CASE eMachineMode OF
	MM_Stopped:
		bAllowDoorsControl := TRUE;
		sModeMask.bRun := FALSE;
		sModeMask.bDashboard := FALSE;
		sModeMask.bManual := TRUE;
		sModeMask.bInit := bLoaderDoorsLocked AND bPearlingDoorsLocked AND NOT bInError;
		sModeMask.bStop := FALSE;
		sModeMask.bPurge := FALSE;
		sModeMask.bPause := FALSE;
		bCanChangeTool := sModeMask.bInit;
		bDoChangeTool := FALSE;
		IF sModeReq.bInit THEN
			eMachineMode := MM_Init;
		END_IF
		IF sModeReq.bManual THEN
			eMachineMode := MM_Manual;
		END_IF
		IF bChangeToolReq AND  eMachineMode = MM_Stopped AND bCanChangeTool THEN
			bDoChangeTool := TRUE;
			eMachineMode := MM_Init;
		END_IF
	MM_Init :
		bAllowDoorsControl := FALSE;
		sModeMask.bRun := FALSE;
		sModeMask.bDashboard := FALSE;
		sModeMask.bManual := FALSE;
		sModeMask.bInit := FALSE;
		sModeMask.bStop := FALSE;
		sModeMask.bPurge := FALSE;
		sModeMask.bPause := FALSE;
		IF bDoChangeTool THEN
			bCanChangeTool := bBlinking;
		ELSE
			bCanChangeTool := TRUE;
			IF bChangeToolReq THEN
				bDoChangeTool := TRUE;
			END_IF
		END_IF
		CASE eStep OF
			SP_RunStp0 : (* Init TurnOver / Pearling / Utilities*)
				eCmdTurnOver := MC_Init;
				eCmdUtilities := MC_Init;
				eCmdPearling := MC_Init;
				eStep := SP_RunStp1;
			SP_RunStp1:
				IF (sMachineData.sModTurnOver.eStatus = MS_Ready) AND (sMachineData.sModPearling.eStatus = MS_Ready) AND (sMachineData.sModUtilities.eStatus = MS_Ready) THEN
					// Init Loader / Barrel / sharpen
					eCmdLoader := MC_Init;
					eCmdBarrel := MC_Init;
					eCmdSharpen := MC_Init;
					eCmdLift1 := MC_Init;
					eCmdLift2 := MC_Init;
					eCmdReject := MC_Init;
					eStep := SP_RunStp2;
				END_IF
				IF (sMachineData.sModTurnOver.eStatus = MS_Stopped) OR  (sMachineData.sModPearling.eStatus = MS_Stopped) OR  (sMachineData.sModUtilities.eStatus = MS_Stopped) THEN
					eMachineMode := MM_ForceStop;
				END_IF
			SP_RunStp2:
				IF (sMachineData.sModLoader.eStatus = MS_Ready) AND (sMachineData.sModBarrel.eStatus = MS_Ready) AND (sMachineData.sModSharpen.eStatus = MS_Ready) THEN
					eCmdTable := MC_Init;
(*					eCmdLift1 := MC_Init;
					eCmdLift2 := MC_Init;
					eCmdReject := MC_Init;*)
					eCmdVision := MC_Init;
					eStep := SP_RunStp3;
				END_IF
				IF (sMachineData.sModLoader.eStatus = MS_Stopped) OR  (sMachineData.sModBarrel.eStatus = MS_Stopped) OR  (sMachineData.sModSharpen.eStatus = MS_Stopped) THEN
					eMachineMode := MM_ForceStop;
				END_IF
			SP_RunStp3 : (* Leave Init *)
				IF bAllModuleInReady THEN
					eMachineMode := MM_Ready;
				END_IF
				IF bOneModuleInStop THEN
					eMachineMode := MM_ForceStop;
				END_IF
		END_CASE
	MM_Ready:
		bAllowDoorsControl := TRUE;
		sModeMask.bRun := bJobInProgress AND NOT bVisionInConfig;
		sModeMask.bDashboard := TRUE;
		sModeMask.bManual := TRUE;
		sModeMask.bInit := FALSE;
		sModeMask.bStop := TRUE;
		sModeMask.bPurge := FALSE;
		sModeMask.bPause := FALSE;
		IF bDoChangeTool THEN
			bCanChangeTool := bBlinking;
		ELSE
			bCanChangeTool := TRUE;
			IF bChangeToolReq THEN
				bDoChangeTool := TRUE;
			END_IF
		END_IF
		IF sModeReq.bRun THEN eMachineMode := MM_Running; END_IF
		IF sModeReq.bDashboard THEN eMachineMode := MM_Dashboard; END_IF
		IF sModeReq.bManual THEN eMachineMode := MM_Manual; END_IF
		IF sModeReq.bStop THEN eMachineMode := MM_ForceStop; END_IF
		IF bOneModuleInStop THEN
			eMachineMode := MM_ForceStop;
		END_IF
		IF bDoChangeTool THEN
			IF eMachineMode = MM_Ready THEN
				eMachineMode := MM_Dashboard;
			ELSE
				bDoChangeTool := FALSE;
			END_IF
		END_IF
		CASE eStep OF
			SP_RunStp0:
				TReadyToStopTimer(IN:= FALSE);
			SP_RunStp1:
				TReadyToStopTimer(IN:=TRUE, PT:=t#10m);
				IF TReadyToStopTimer.Q AND eMachineMode = MM_Ready THEN
					eMachineMode := MM_ForceStop;
				END_IF
		END_CASE
	MM_Running,MM_Purging :
		bAllowDoorsControl := FALSE;
		sModeMask.bRun := FALSE;
		sModeMask.bDashboard := FALSE;
		sModeMask.bManual := FALSE;
		sModeMask.bInit := FALSE;
		sModeMask.bStop := TRUE;
		sModeMask.bPurge := (eMachineMode = MM_Running) ;
		sModeMask.bPause := TRUE;
		bCanChangeTool := FALSE;
		IF sModeReq.bPause THEN eMachineMode := MM_Pausing; END_IF
		IF sModeReq.bStop THEN eMachineMode := MM_Stopping; END_IF
		IF sModeReq.bPurge THEN
			eMachineMode := MM_Purging;
			eLastMachineMode := eMachineMode;
		END_IF
		CASE eStep OF
			SP_RunStp0:
				eCmdAll := MC_Run;
				bRunInit := TRUE;
				eStep := SP_RunStp1;
			SP_RunStp1:
				IF bRunTestMode THEN
					TManagerRunTest(
						sRunData := sRunData,
						bFirstCycle := bRunInit,
						sConfigFileData := sConfigFileData,
					);
					bRunInit := FALSE;
					sProductionCmd.TRequestSample.Activate := FALSE;
					sProductionCmd.TRequestSample.Enable := FALSE;
				ELSE
					TManagerRun(
						bSimPearling := bSimPearling,
						bPurging := (eMachineMode = MM_Purging) ,
						bFirstCycle := bRunInit,
						sRunData := sRunData,
						sConfigFileData := sConfigFileData,
						sProdLot	 := sProdLot,
						bLayeringWithTwoParts := bLayeringWithTwoParts,
						bNewJob := bNewJobForRun,
						sProductionCmd := sProductionCmd,
						bDisableCleanAfterPearling := bDisableCleanAfterPearling
					);
					bRunInit := FALSE;
					bNewJobForRun := FALSE;
					IF bOneModuleInPause OR bOneModuleInReadyOrStop THEN
						bComputeMTBF := TRUE;
					END_IF
				END_IF
				IF bOneModuleInPause THEN eMachineMode := MM_Pausing; END_IF
				IF bOneModuleInReadyOrStop THEN eMachineMode := MM_Stopping; END_IF
				IF NOT bRunTestMode AND TManagerRun.bRecipeIsFinish THEN eMachineMode := MM_Stopping; END_IF
		END_CASE
	MM_Dashboard:
		bAllowDoorsControl := TRUE;
		sModeMask.bRun := FALSE;
		sModeMask.bDashboard := FALSE;
		sModeMask.bManual := FALSE;
		sModeMask.bInit := FALSE;
		sModeMask.bStop := TRUE;
		sModeMask.bPurge := FALSE;
		sModeMask.bPause := FALSE;
		IF bDoChangeTool THEN
			bCanChangeTool := bBlinking;
		ELSE
			bCanChangeTool := TRUE;
			IF bChangeToolReq THEN
				bDoChangeTool := TRUE;
			END_IF
		END_IF
		IF sModeReq.bStop THEN eMachineMode := MM_Stopping; END_IF
		CASE eStep OF
			SP_RunStp0:
				eCmdAll := MC_Run;
				eStep := SP_RunStp1;
			SP_RunStp1:
				IF bOneModuleInPause THEN eMachineMode := MM_Pausing; END_IF
				IF bOneModuleInReadyOrStop THEN eMachineMode := MM_Stopping; END_IF
		END_CASE
		IF eMachineMode <> MM_Dashboard THEN bDoChangeTool := FALSE; END_IF
	MM_Manual :
		bAllowDoorsControl := TRUE;
		sModeMask.bRun := FALSE;
		sModeMask.bDashboard := FALSE;
		sModeMask.bManual := FALSE;
		sModeMask.bInit := bLoaderDoorsLocked AND bPearlingDoorsLocked AND NOT bInError;
		sModeMask.bStop := TRUE;
		sModeMask.bPurge := FALSE;
		sModeMask.bPause := FALSE;
		bCanChangeTool := FALSE;
		IF sModeReq.bStop THEN eMachineMode := MM_Stopping; END_IF
		IF sModeReq.bInit THEN
			eMachineMode := MM_Stopping;
			bDoInitAfterStop := TRUE;
		END_IF
		CASE eStep OF
			SP_RunStp0:
				eCmdAll := MC_Manual;
				eStep := SP_RunStp1;
			SP_RunStp1:
				eStep := SP_RunStp1;
		END_CASE;
	MM_Stopping:
		bAllowDoorsControl := FALSE;
		sModeMask.bRun := FALSE;
		sModeMask.bDashboard := FALSE;
		sModeMask.bManual := FALSE;
		sModeMask.bInit := FALSE;
		sModeMask.bStop := TRUE;
		sModeMask.bPurge := FALSE;
		sModeMask.bPause := FALSE;
		bCanChangeTool := FALSE;
		CASE eStep OF
			SP_RunStp0:
				TForceStop(IN := FALSE);
				eStep := SP_RunStp1;
			SP_RunStp1:
				TForceStop(IN := TRUE, PT := TMaxStopppingTime);
				IF bAllModuleInReady THEN
					IF TManagerRun.bRecipeIsFinish THEN
						eMachineMode := MM_Stopped;
						eCmdUtilities := MC_Stop;
					ELSE
						eMachineMode := MM_Ready;
					END_IF
					bDoInitAfterStop := FALSE;
				ELSIF bAllModuleInReadyOrStop AND bOneModuleInStop THEN
					IF bDoInitAfterStop AND bLoaderDoorsLocked AND bPearlingDoorsLocked AND NOT bInError THEN
						eMachineMode := MM_Init;
					ELSE
						eMachineMode := MM_Stopped;
					END_IF
					bDoInitAfterStop := FALSE;
				ELSIF TForceStop.Q OR sModeReq.bStop  THEN
					eMachineMode := MM_ForceStop;
				END_IF
		END_CASE;
	MM_ForceStop:
		bAllowDoorsControl := FALSE;
		sModeMask.bRun := FALSE;
		sModeMask.bDashboard := FALSE;
		sModeMask.bManual := FALSE;
		sModeMask.bInit := FALSE;
		sModeMask.bStop := FALSE;
		sModeMask.bPurge := FALSE;
		sModeMask.bPause := FALSE;
		bCanChangeTool := FALSE;
		CASE eStep OF
			SP_RunStp0:
				eCmdAll := MC_Stop;
				eStep := SP_RunStp1;
			SP_RunStp1:
				IF bAllModuleInStop THEN
					IF bDoInitAfterStop AND bLoaderDoorsLocked AND bPearlingDoorsLocked AND NOT bInError THEN
						eMachineMode := MM_Init;
					ELSE
						eMachineMode := MM_Stopped;
					END_IF
					bDoInitAfterStop := FALSE;
				END_IF
		END_CASE;
	MM_Pausing:
		bAllowDoorsControl := FALSE;
		sModeMask.bRun := FALSE;
		sModeMask.bDashboard := FALSE;
		sModeMask.bManual := FALSE;
		sModeMask.bInit := FALSE;
		sModeMask.bStop := TRUE;
		sModeMask.bPurge := FALSE;
		sModeMask.bPause := FALSE;
		bCanChangeTool := FALSE;
		CASE eStep OF
			SP_RunStp0:
				TForceStop(IN := FALSE);
				eStep := SP_RunStp1;
			SP_RunStp1:
				TForceStop(IN := TRUE, PT := TMaxPausingTime);
				IF bAllModuleInPause THEN
					eMachineMode := MM_Pause;
				ELSIF TForceStop.Q OR sModeReq.bStop OR bOneModuleInReadyOrStop  THEN
					eMachineMode := MM_Stopping;
				END_IF
		END_CASE;
	MM_Pause:
		bAllowDoorsControl := TRUE;
		sModeMask.bRun := TRUE;
		sModeMask.bDashboard := FALSE;
		sModeMask.bManual := TRUE;
		sModeMask.bInit := FALSE;
		sModeMask.bStop := TRUE;
		sModeMask.bPurge := FALSE;
		sModeMask.bPause := FALSE;
		bCanChangeTool := FALSE;
		IF sModeReq.bRun THEN eMachineMode := MM_Running; END_IF
		IF sModeReq.bManual THEN eMachineMode := MM_Manual; END_IF
		IF sModeReq.bStop THEN eMachineMode := MM_Stopping; END_IF
		IF bOneModuleInReadyOrStop THEN
			eMachineMode := MM_Stopping;
		END_IF
END_CASE;

TManagerDashboard(
	bExecute := eMachineMode = MM_Dashboard AND eLastMachineMode = eMachineMode AND eStep = SP_RunStp1,
	sRunData := sRunData,
	bDoChangeTool := bDoChangeTool,
	sConfigFileData := sConfigFileData,
	sCmd := sDashboardCmd
);

bInJobMode := ((eMachineMode = MM_Running) OR (eMachineMode = MM_Purging)) AND eLastMachineMode = eMachineMode AND eStep = SP_RunStp1 AND NOT bRunTestMode;
TJobElapsedCounter(
	bRun := bInJobMode,
	bReset := FALSE,
	bSet := FALSE
	);
TMTBFCounter(
	bStart := bInJobMode,
	bReset := FALSE
	);
IF bComputeMTBF THEN
	bComputeMTBF := FALSE;
	iMTBFCounter := iMTBFCounter + 1;
	dwMTBFTotalTime := dwMTBFTotalTime + TMTBFCounter.dwSeconds;
	TMTBFCounter(
		bReset := TRUE
		);
END_IF
IF bResetMTBF THEN
	bResetMTBF := FALSE;
	dwMTBFTotalTime := 0;
	iMTBFCounter := 0;
END_IF
IF iMTBFCounter > 0 THEN
	dwMeanMTBF := dwMTBFTotalTime / INT_TO_DWORD(iMTBFCounter);
ELSE
	dwMeanMTBF := 0;
END_IF

(* Running time counters *)
TMachineOnCounter(bStart := TRUE, bReset := bResetMachineCounters);
TInProdCounter(bStart := (eMachineMode = MM_Running) OR (eMachineMode = MM_Purging), bReset := bResetMachineCounters);

(* Clear  mode requests *)
sModeReq.bStop := FALSE;
sModeReq.bInit := FALSE;
sModeReq.bManual := FALSE;
sModeReq.bRun := FALSE;
sModeReq.bPurge := FALSE;
sModeReq.bPause := FALSE;
sModeReq.bDashboard := FALSE;


IF eCmdAll<> MC_NoCmd THEN
	eCmdLoader := eCmdAll;
	eCmdTable:= eCmdAll;
	eCmdPearling := eCmdAll;
	eCmdTurnOver := eCmdAll;
	eCmdBarrel := eCmdAll;
	eCmdSharpen := eCmdAll;
	eCmdLift1 := eCmdAll;
	eCmdLift2 := eCmdAll;
	eCmdReject := eCmdAll;
	eCmdVision := eCmdAll;
	eCmdUtilities := eCmdAll;
END_IF

TWritePersistentData(
	PORT    := 852,
	START := bSavePersistent,
	MODE    := SPDM_2PASS
);

IF bNewJob  THEN
	bJobInProgress := TRUE;
	bNewJobForRun := TRUE;
	TJobElapsedCounter(
		bRun := FALSE,
		bReset := FALSE,
		bSet := TRUE,
		tSetTime := DWORD_TO_TIME(dwStartJobElapsedTime)
	);
END_IF
IF bEndOfJob THEN
	bJobInProgress := FALSE;
	TJobElapsedCounter(
		bRun := FALSE,
		bReset := TRUE,
		bSet := FALSE
	);
END_IF
TJobElapsed := TJobElapsedCounter.TElapsed;

dwJobQty := sProdLot.dLotQty;
IF eMachineMode = MM_Purging THEN
	IF C_PROD_MODE_GOOD_PART THEN
		dwJobQty := sProdLot.dGoodQty + (sProdLot.dLoadedQty - sProdLot.dProdQty);
	ELSE
		dwJobQty := sProdLot.dLoadedQty;
	END_IF
END_IF

IF sProdLot.dEstimatedPartTime*dwJobQty > TIME_TO_DWORD(TJobElapsed) THEN
	dwProdEstimatedTimeLeft := sProdLot.dEstimatedPartTime*dwJobQty - TIME_TO_DWORD(TJobElapsed);
ELSE
	dwProdEstimatedTimeLeft := 0;
END_IF

IF NOT TWritePersistentData.BUSY AND bSavePersistent THEN
	bSavePersistent := FALSE;
END_IF

IF eMachineMode <> MM_Running AND  eMachineMode <> MM_Purging THEN
	sProductionCmd.TRequestSample.Enable := FALSE;
	sProductionCmd.TRequestSample.Activate := FALSE;
END_IF


IF eMachineMode = MM_Dashboard THEN
	eManagerRunStep := TManagerDashboard.eManagerStep;
ELSE
	IF bRunTestMode THEN
		eManagerRunStep := TManagerRunTest.eManagerStep;
	ELSE
		eManagerRunStep := TManagerRun.eManagerStep;
	END_IF
END_IF

bReadyForChangeJob := (eMachineMode = MM_Stopped);
bStopRequest := (eMachineMode = MM_Stopping);
bPauseRequest := (eMachineMode = MM_Pausing);
bPearlingHead1IsUsed := (sConfigFileData.asPearlingData[PS_SUS].THead[PH_Left].nNbOfPearls > 0) OR (sConfigFileData.asPearlingData[PS_SOUS].THead[PH_Left].nNbOfPearls > 0);
bPearlingHead2IsUsed := (sConfigFileData.asPearlingData[PS_SUS].THead[PH_Right].nNbOfPearls > 0) OR (sConfigFileData.asPearlingData[PS_SOUS].THead[PH_Right].nNbOfPearls > 0);
bLayeringWithTwoParts := ((sConfigFileData.sPartData.alrPartOffsetLayering[1].lrX <> 0) OR (sConfigFileData.sPartData.alrPartOffsetLayering[1].lrY <> 0));
bConfigError := TManagerRun.bConfigError;

(* MDE option *)
IF bFillMDE THEN
	(* Update MDE *)
	TMDEData.dwPceGood := sMachineData.sCounter.sProd.dGood;
	TMDEData.dwPceBad := sMachineData.sCounter.sProd.dTotal  - TMDEData.dwPceGood;
	
	(* MDE status *)
	IF bInError THEN
		TMDEData.iStatus := MDE_Alarm;
	ELSIF (eMachineMode = MM_Running) THEN
		TMDEData.iStatus := MDE_Production;
	ELSIF (eMachineMode = MM_Manual) THEN
		TMDEData.iStatus := MDE_Maintenance;
	ELSE
		TMDEData.iStatus := MDE_Standby;
	END_IF
	(* MDE alarm *)
	TMDEData.iPertCode := iMDEAlarm;
END_IF

END_FUNCTION_BLOCK

// ---- POUs/utils/HandleErrors.TcPOU
FUNCTION_BLOCK HandleErrors
VAR_INPUT
	bEnable					: BOOL;
(*	bUsingLeft				: BOOL;
	bUsingRight				: BOOL;*)
	abErrorsTable			: ARRAY[0..C_MAX_NB_OF_ERRORS] OF BOOL;
END_VAR
VAR_OUTPUT
	bInError					: BOOL;
	bInWarning				: BOOL;
	iMDEAlarm				: INT;
END_VAR
VAR_IN_OUT
END_VAR
VAR
END_VAR

bInError :=
	abErrorsTable[ERR_Manager]
	OR abErrorsTable[ERR_EmergencyStop]
	OR abErrorsTable[ERR_AirPressure]
	OR abErrorsTable[ERR_24VPowerSupply]
	OR abErrorsTable[ERR_48VPowerSupply]
	OR abErrorsTable[ERR_DrivesAreOFF]
	OR abErrorsTable[ERR_Aspiration]
	OR abErrorsTable[ERR_LoaderAxisX]
	OR abErrorsTable[ERR_LoaderAxisY]
	OR abErrorsTable[ERR_LoaderAxisZ1]
	OR abErrorsTable[ERR_LoaderAxisZ2]
	OR abErrorsTable[ERR_LoaderAxisTheta]
	OR abErrorsTable[ERR_LoaderHead1Vacuum]
	OR abErrorsTable[ERR_LoaderHead2Vacuum]
	OR abErrorsTable[ERR_LoaderJack]
	OR abErrorsTable[ERR_LoaderPlateVacuum]
	OR abErrorsTable[ERR_LoaderVision]
	OR abErrorsTable[ERR_LoaderNoPartTaken]
	OR abErrorsTable[ERR_Lift1Drv]
	OR abErrorsTable[ERR_Lift2Drv]
	OR abErrorsTable[ERR_BarrelAxis]
	OR abErrorsTable[ERR_BarrelJack]
	OR abErrorsTable[ERR_BarrelIndex]
	OR abErrorsTable[ERR_BarrelStickNotTaken]
	OR abErrorsTable[ERR_BarrelEmpty]
	OR abErrorsTable[ERR_PearlingAxisX]
	OR abErrorsTable[ERR_PearlingAxisY]
	OR abErrorsTable[ERR_PearlingAxisZ1]
	OR abErrorsTable[ERR_PearlingAxisZ2]
	OR abErrorsTable[ERR_PearlingSpindle1]
	OR abErrorsTable[ERR_PearlingSpindle2]
	OR abErrorsTable[ERR_PearlingGripper1]
	OR abErrorsTable[ERR_PearlingGripper2]
	OR abErrorsTable[ERR_PearlingMCR]
	OR abErrorsTable[ERR_PearlingSecurity]
	OR abErrorsTable[ERR_TableAxis]
	OR abErrorsTable[ERR_TablePearlingAspiration]
	OR abErrorsTable[ERR_TableJack]
	OR abErrorsTable[ERR_TablePos1Vacuum]
	OR abErrorsTable[ERR_TablePos2Vacuum]
	OR abErrorsTable[ERR_TablePos3Vacuum]
	OR abErrorsTable[ERR_TablePos4Vacuum]
	OR abErrorsTable[ERR_TableVacuum4Rotation]
	OR abErrorsTable[ERR_PearlingMotor1]
	OR abErrorsTable[ERR_PearlingMotor2]
	OR abErrorsTable[ERR_PearlingCurrent1]
	OR abErrorsTable[ERR_PearlingCurrent2]
	OR abErrorsTable[ERR_BrushAxis]
	OR abErrorsTable[ERR_SharpenAxis]
	OR abErrorsTable[ERR_SharpenTape]
	OR abErrorsTable[ERR_TurnOverAxis]
	OR abErrorsTable[ERR_TurnOverJack]
	OR abErrorsTable[ERR_TurnOverArmVacuum]
	OR abErrorsTable[ERR_TurnOverFixVacuum]
	OR abErrorsTable[ERR_VisionNotReady]
	OR abErrorsTable[ERR_VisionNotConnected]
	OR abErrorsTable[ERR_Vacuum]
	OR abErrorsTable[ERR_LoaderZSensorOutOfRange]
	OR abErrorsTable[ERR_RejectDrawerOpened]
	OR abErrorsTable[ERR_ConfigNotUsable]
	OR abErrorsTable[ERR_Lift1PlateLock]
	OR abErrorsTable[ERR_Lift1DrawerLock]
	OR abErrorsTable[ERR_Lift2PlateLock]
	OR abErrorsTable[ERR_Lift2DrawerLock]
	OR abErrorsTable[ERR_TableCleanBrush]
	
;

bInWarning :=
	abErrorsTable[W_LoaderDoorsNotClosed]
	OR abErrorsTable[W_PearlingDoorsNotClosed]
	OR abErrorsTable[W_NoPowerOnV1]
	OR abErrorsTable[W_DoorsNotLocked]
	OR abErrorsTable[W_LoaderSamplesReady]
	OR abErrorsTable[W_RejectChangePlate]
	OR abErrorsTable[W_Lift1NeedPlate]
	OR abErrorsTable[W_Lift2NeedPlate]
	OR abErrorsTable[W_Lift1DrawerNotInPos]
	OR abErrorsTable[W_Lift2DrawerNotInPos]
	OR abErrorsTable[W_RejectDrawerNotInPos]
	OR abErrorsTable[W_RejectPlateNotInPos]
	OR abErrorsTable[W_BarrelNeedArea1Stick]
	OR abErrorsTable[W_BarrelNeedArea2Stick]
	OR abErrorsTable[W_BarrelNeedArea3Stick]
	OR abErrorsTable[W_BarrelNeedArea4Stick]
	OR abErrorsTable[W_JobPurged]
	OR abErrorsTable[W_LoaderPartsOnPlate]
	OR abErrorsTable[W_VisionInSimulation]
	OR abErrorsTable[W_Lift1BadPlate]
	OR abErrorsTable[W_PearlingLeftStickBroken]
	OR abErrorsTable[W_PearlingRightStickBroken]
	OR abErrorsTable[W_PearlingWeight1OutOfTolerance]
	OR abErrorsTable[W_PearlingWeight2OutOfTolerance]
	OR abErrorsTable[W_PearlingLeftSpindleUsed]
	OR abErrorsTable[W_PearlingRightSpindleUsed]
	OR abErrorsTable[W_PearlingLeftMotorUsed]
	OR abErrorsTable[W_PearlingRightMotorUsed]
	OR abErrorsTable[W_PearlingLeftSpindleLimit]
	OR abErrorsTable[W_PearlingRightSpindleLimit]
	OR abErrorsTable[W_PearlingLeftSpindleHeat]
	OR abErrorsTable[W_PearlingRightSpindleHeat]
;
(* Handle TMDE error status *)
IF bInError THEN
	(* Update alarm status only if not already set *)
	IF (iMDEAlarm = 2900) OR (iMDEAlarm = 0) THEN
		(* Define code depending on alarm *)
		IF abErrorsTable[ERR_ConfigNotUsable]
				OR abErrorsTable[ERR_Aspiration]
				OR abErrorsTable[ERR_VisionNotReady]
				OR abErrorsTable[ERR_VisionNotConnected]
			THEN
			iMDEAlarm := 2010; 		(* General alarm*)
		ELSIF abErrorsTable[ERR_24VPowerSupply]
				OR abErrorsTable[ERR_48VPowerSupply]
				OR abErrorsTable[ERR_DrivesAreOFF]  THEN
			iMDEAlarm := 2020; 		(* Electrial alarm*)
		ELSIF abErrorsTable[ERR_LoaderAxisX]
				OR abErrorsTable[ERR_LoaderAxisY]
				OR abErrorsTable[ERR_LoaderAxisZ1]
				OR abErrorsTable[ERR_LoaderAxisZ2]
				OR abErrorsTable[ERR_LoaderAxisTheta]
				OR abErrorsTable[ERR_Lift1Drv]
				OR abErrorsTable[ERR_Lift2Drv]
				OR abErrorsTable[ERR_PearlingAxisX]
				OR abErrorsTable[ERR_PearlingAxisY]
				OR abErrorsTable[ERR_PearlingAxisZ1]
				OR abErrorsTable[ERR_PearlingAxisZ2]
				OR abErrorsTable[ERR_BarrelAxis]
				OR abErrorsTable[ERR_TableAxis]
				OR abErrorsTable[ERR_SharpenAxis]
				OR abErrorsTable[ERR_TurnOverAxis]
				OR abErrorsTable[ERR_BrushAxis]
				THEN
			iMDEAlarm := 2021; 		(* Motor alarm*)
		ELSIF abErrorsTable[ERR_RejectDrawerOpened]
				OR abErrorsTable[ERR_PearlingSecurity]
				OR abErrorsTable[ERR_TablePearlingAspiration]
				OR abErrorsTable[ERR_TableJack]
				OR abErrorsTable[ERR_BarrelJack]
				OR abErrorsTable[ERR_BarrelIndex]
				OR abErrorsTable[ERR_TurnOverJack]
				OR abErrorsTable[ERR_LoaderZSensorOutOfRange]
				OR abErrorsTable[ERR_LoaderJack]
				OR abErrorsTable[ERR_Lift1PlateLock]
				OR abErrorsTable[ERR_Lift1DrawerLock]
				OR abErrorsTable[ERR_Lift2PlateLock]
				OR abErrorsTable[ERR_Lift2DrawerLock]
				OR abErrorsTable[ERR_TableCleanBrush]
				THEN
			iMDEAlarm := 2040; 		(* Machine security alarm*)
		ELSIF abErrorsTable[ERR_EmergencyStop]
				THEN
			iMDEAlarm := 2050; 		(* Human security alarm*)
		ELSIF abErrorsTable[ERR_PearlingMCR]
				OR abErrorsTable[ERR_PearlingGripper1]
				OR abErrorsTable[ERR_PearlingGripper2]
				OR abErrorsTable[ERR_PearlingSpindle1]
				OR abErrorsTable[ERR_PearlingSpindle2]
				OR abErrorsTable[ERR_SharpenTape]
				THEN
			iMDEAlarm := 2060; 		(* General tool alarm*)
		ELSIF	abErrorsTable[ERR_AirPressure]
				THEN
			iMDEAlarm := 2070; 		(* Pneumatics alarm*)
		ELSIF FALSE THEN
			iMDEAlarm := 2100; 		(* Power down alarm*)
		ELSIF FALSE THEN
			iMDEAlarm := 2101; 		(* Init alarm*)
		ELSIF FALSE THEN
			iMDEAlarm := 2102; 		(* Warming alarm*)
		ELSIF FALSE THEN
			iMDEAlarm := 2103; 		(* Ready for prod alarm*)
		ELSIF abErrorsTable[ERR_BarrelEmpty] THEN
			iMDEAlarm := 2110; 		(* Material supply alarm*)
		ELSIF FALSE THEN
			iMDEAlarm := 2121; 		(* NbOfParts reached alarm*)
		ELSIF abErrorsTable[ERR_LoaderHead1Vacuum]
				OR abErrorsTable[ERR_LoaderHead2Vacuum]
				OR abErrorsTable[ERR_TablePos1Vacuum]
				OR abErrorsTable[ERR_TablePos2Vacuum]
				OR abErrorsTable[ERR_TablePos3Vacuum]
				OR abErrorsTable[ERR_TablePos4Vacuum]
				OR abErrorsTable[ERR_TurnOverArmVacuum]
				OR abErrorsTable[ERR_TurnOverFixVacuum]
				OR abErrorsTable[ERR_TableVacuum4Rotation]
				OR abErrorsTable[ERR_PearlingMotor1]
				OR abErrorsTable[ERR_PearlingMotor2]
				OR abErrorsTable[ERR_PearlingCurrent1]
				OR abErrorsTable[ERR_PearlingCurrent2]
				OR abErrorsTable[ERR_BarrelStickNotTaken]
				OR abErrorsTable[ERR_LoaderPlateVacuum]
				OR abErrorsTable[ERR_Vacuum]
				THEN
			iMDEAlarm := 2200; 		(* Process alarm*)
		ELSIF FALSE THEN
			iMDEAlarm := 2312; 		(* Tools alarm*)
		ELSE
			iMDEAlarm := 2010; 		(* By default general alarm*)
		END_IF
	END_IF
ELSIF binWarning THEN
	iMDEAlarm := 2900;
ELSE
	iMDEAlarm := 0;
END_IF

END_FUNCTION_BLOCK

// ---- POUs/utils/TBlink.TcPOU
FUNCTION_BLOCK TBlink
VAR_INPUT
	bEnable			: BOOL;
	tOnPeriod		: TIME		:= t#500ms;
	tOffPeriod		: TIME		:= t#500ms;
END_VAR
VAR_OUTPUT
	bBlink			: BOOL;
END_VAR
VAR
	TBlinker			: TON;
(*	bBlinkOn			: BOOL;*)
	CurrentPeriod		: TIME		:= t#10ms;
END_VAR

IF bEnable THEN
	TBlinker(IN := TRUE,PT := CurrentPeriod);
ELSE
	TBlinker(IN := FALSE);
END_IF

IF bBlink AND TBlinker.Q THEN
	bBlink := FALSE;
	CurrentPeriod := tOffPeriod;
	TBlinker(IN := FALSE);
ELSIF NOT bBlink AND TBlinker.Q THEN
	bBlink := TRUE;
	CurrentPeriod := tOnPeriod;
	TBlinker(IN := FALSE);
END_IF

END_FUNCTION_BLOCK

// ---- POUs/Manager/ManagerDashboard.TcPOU
FUNCTION_BLOCK ManagerDashboard
VAR_INPUT
	sConfigFileData			: TConfigFileData;
(*	bFirstCycle				: BOOL;*)
	bExecute				: BOOL;
END_VAR
VAR_OUTPUT
END_VAR
VAR_IN_OUT
	bDoChangeTool			: BOOL;
	sRunData				: TRunData;
	sCmd					: TDashboardCmd;
END_VAR
VAR
	eManagerStep			: TModuleSteps := SP_RunStp0;
	bLastExecute				: BOOL;
	iCurrentLift				: INT;
END_VAR

sCmd.iMaxScanModel := sRunData.TDataVision.iMaxModel;
IF NOT bExecute THEN
	sCmd.TLoaderEndOfRecipe.Enable := FALSE;
	sCmd.TLoaderScanPlateLift1.Enable := FALSE;
	sCmd.TLoaderScanPlateLift2.Enable := FALSE;
	sCmd.TLoaderScanPlateReject.Enable := FALSE;
	sCmd.TPickPlace.Enable := FALSE;
	sCmd.TTableTurn.Enable := FALSE;
	sCmd.TPearling.Enable := FALSE;
	sCmd.TLoaderEndOfRecipe.Activate := FALSE;
	sCmd.TLoaderScanPlateLift1.Activate := FALSE;
	sCmd.TLoaderScanPlateLift2.Activate := FALSE;
	sCmd.TLoaderScanPlateReject.Activate := FALSE;
	sCmd.TPickPlace.Activate := FALSE;
	sCmd.TTableTurn.Activate := FALSE;
	sCmd.TPearling.Activate := FALSE;
	bLastExecute := FALSE;
ELSE
	sRunData.eCmdTurnOver := RCTO_None;
	sRunData.eCmdTable := RCT_None;
	sRunData.eCmdLoader := RCLo_None;
	sRunData.eCmdPearling := RCP_None;
	IF bLastExecute = FALSE THEN
		bLastExecute := TRUE;
		eManagerStep := SP_RunStp0;
	END_IF
	sCmd.TLoaderEndOfRecipe.Enable := sRunData.sStatusLoader = RS_WaitRequest AND eManagerStep = SP_RunStp1;
	sCmd.TLoaderScanPlateLift1.Enable := sRunData.sStatusLoader = RS_WaitRequest AND eManagerStep = SP_RunStp1;
	sCmd.TLoaderScanPlateLift2.Enable := sRunData.sStatusLoader = RS_WaitRequest AND eManagerStep = SP_RunStp1;
	sCmd.TLoaderScanPlateReject.Enable := sRunData.sStatusLoader = RS_WaitRequest AND eManagerStep = SP_RunStp1;
	sCmd.TPickPlace.Enable := (sRunData.sStatusLoader = RS_WaitRequest AND sRunData.sStatusTable = RS_WaitRequest AND eManagerStep = SP_RunStp1) OR (eManagerStep >= SP_RunStp30 AND eManagerStep <= SP_RunStp49);
	sCmd.TTableTurn.Enable := sRunData.sStatusLoader = RS_WaitRequest AND sRunData.sStatusTable = RS_WaitRequest AND eManagerStep = SP_RunStp1;
	sCmd.TPearling.Enable := sRunData.sStatusPearling = RS_WaitRequest AND eManagerStep = SP_RunStp1;;
	CASE eManagerStep OF
		SP_RunStp0:
			sCmd.TLoaderEndOfRecipe.Activate := FALSE;
			sCmd.TLoaderScanPlateLift1.Activate := FALSE;
			sCmd.TLoaderScanPlateLift2.Activate := FALSE;
			sCmd.TLoaderScanPlateReject.Activate := FALSE;
			sCmd.TPickPlace.Activate := FALSE;
			sCmd.TTableTurn.Activate := FALSE;
			sCmd.TPearling.Activate := FALSE;
			eManagerStep := SP_RunStp1;
		SP_RunStp1:
			IF sCmd.TLoaderEndOfRecipe.Activate THEN
				sCmd.TLoaderEndOfRecipe.Activate := FALSE;
				sRunData.eCmdLoader := RCLo_EndOfRecipe;
				eManagerStep := SP_RunStp10;
			END_IF
			IF sCmd.TLoaderScanPlateLift1.Activate THEN
				sCmd.TLoaderScanPlateLift1.Activate := FALSE;
				sRunData.TDataLoader.eModule := LMP_Lift1;
				sRunData.TDataLoader.iScanModel := sCmd.iScanModel;
				sRunData.eCmdLoader := RCLo_ScanPlate;
				iCurrentLift := 0;
				eManagerStep := SP_RunStp5;
			END_IF
			IF sCmd.TLoaderScanPlateLift2.Activate THEN
				sCmd.TLoaderScanPlateLift2.Activate := FALSE;
				sRunData.TDataLoader.eModule := LMP_Lift2;
				sRunData.TDataLoader.iScanModel := sCmd.iScanModel;
				sRunData.eCmdLoader := RCLo_ScanPlate;
				iCurrentLift := 1;
				eManagerStep := SP_RunStp5;
			END_IF
			IF sCmd.TLoaderScanPlateReject.Activate THEN
				sCmd.TLoaderScanPlateReject.Activate := FALSE;
				sRunData.TDataLoader.eModule := LMP_Reject;
				sRunData.TDataLoader.iScanModel := sCmd.iScanModel;
				sRunData.eCmdLoader := RCLo_ScanPlate;
				iCurrentLift := 2;
				eManagerStep := SP_RunStp5;
			END_IF
			IF sCmd.TTableTurn.Activate THEN
				sCmd.TTableTurn.Activate := FALSE;
				eManagerStep := SP_RunStp20;
			END_IF
			IF sCmd.TPickPlace.Activate THEN
				eManagerStep := SP_RunStp30;
			END_IF
			IF sCmd.TPearling.Activate OR bDoChangeTool THEN
				bDoChangeTool := TRUE;
				sCmd.TPearling.Activate := FALSE;
				sRunData.eCmdPearling := RCP_ChangeChuck;
				eManagerStep := SP_RunStp50;
			END_IF
		SP_RunStp5:
			(* Update scan data *)
			sCmd.aiScanPlateOK[iCurrentLift] := sRunData.TDataLoader.iCurrentScanOK;
			sCmd.aiScanPlateTotal[iCurrentLift] := sRunData.TDataLoader.iCurrentScanTotal;
			IF sRunData.sStatusLoader = RS_WaitRequest THEN
				eManagerStep := SP_RunStp1;
			END_IF
		SP_RunStp10:
			IF sRunData.sStatusLoader = RS_WaitRequest THEN
				eManagerStep := SP_RunStp1;
			END_IF
		SP_RunStp20:
			sRunData.eCmdLoader := RCLo_MoveToSafe;
			eManagerStep := SP_RunStp21;
		SP_RunStp21:
			IF sRunData.sStatusLoader = RS_WaitRequest THEN
				sRunData.eCmdTable := RCT_Turn;
				eManagerStep := SP_RunStp22;
			END_IF
		SP_RunStp22:
			IF sRunData.sStatusLoader = RS_WaitRequest AND  sRunData.sStatusTable = RS_WaitRequest THEN
				eManagerStep := SP_RunStp1;
			END_IF
		SP_RunStp30: (* Unloading part on layering 0 *)
			IF NOT sCmd.TPickPlace.Activate THEN
				eManagerStep := SP_RunStp1;(* End *)
			ELSIF sRunData.TDataTable.aTPartData[0,0,sRunData.TDataTable.eTableSide].bPartPresent THEN
				eManagerStep := SP_RunStp31;
			ELSE
				eManagerStep := SP_RunStp40;(* Skip *)
			END_IF
		SP_RunStp31:
			sRunData.TDataLoader.eModule := LMP_Table;
			sRunData.TDataLoader.eTaker := LH_Head1;
			sRunData.TDataLoader.iLayringPos := 0;
			sRunData.TDataLoader.iLayringOffsetPos := 0;
			sRunData.eCmdLoader := RCLo_PrepareTakePart;
			eManagerStep := SP_RunStp32;
		SP_RunStp32:
			IF sRunData.sStatusLoader = RS_WaitRequest THEN
				sRunData.eCmdLoader := RCLo_TakePart;
				sRunData.TDataTable.iGiveTakeLayeringPosition := sRunData.TDataLoader.iLayringPos;
				sRunData.TDataTable.iGiveTakeLayeringOffsetPosition := sRunData.TDataLoader.iLayringOffsetPos;
				sRunData.eCmdTable := RCT_GivePart;
				eManagerStep := SP_RunStp33;
			END_IF
		SP_RunStp33:
			IF sRunData.sStatusLoader = RS_WaitRequest AND  sRunData.sStatusTable = RS_WaitRequest  THEN
				sRunData.TDataLoader.eModule := LMP_Lift2;
				sRunData.eCmdLoader := RCLo_PrepareDropPart;
				eManagerStep := SP_RunStp35;
			END_IF
		SP_RunStp35:
			IF sRunData.sStatusLoader = RS_WaitRequest THEN
				sRunData.eCmdLoader := RCLo_GivePart;
				eManagerStep := SP_RunStp36;
			END_IF
		SP_RunStp36:
			IF sRunData.sStatusLoader = RS_WaitRequest THEN
				eManagerStep := SP_RunStp40;
			END_IF
		SP_RunStp40: (* Load layering 1 *)
			IF NOT sCmd.TPickPlace.Activate THEN
				eManagerStep := SP_RunStp1;(* End *)
			ELSIF NOT sRunData.TDataTable.aTPartData[0,0,sRunData.TDataTable.eTableSide].bPartPresent THEN
				sRunData.TDataLoader.eModule := LMP_Lift1;
				sRunData.TDataLoader.eTaker := LH_Head1;
				sRunData.eCmdLoader := RCLo_PrepareTakePart;
				eManagerStep := SP_RunStp41;
			ELSE
				eManagerStep := SP_RunStp30;(* Skip *)
			END_IF
		SP_RunStp41:
			IF sRunData.sStatusLoader = RS_WaitRequest THEN
				sRunData.eCmdLoader := RCLo_TakePart;
				eManagerStep := SP_RunStp42;
			END_IF
		SP_RunStp42:
			IF sRunData.sStatusLoader = RS_WaitRequest THEN
				sRunData.TDataLoader.eModule := LMP_Table;
				sRunData.TDataLoader.iLayringPos := 0;
				sRunData.TDataLoader.iLayringOffsetPos := 0;
				sRunData.eCmdLoader := RCLo_PrepareDropPart;
				eManagerStep := SP_RunStp43;
			END_IF
		SP_RunStp43:
			IF sRunData.sStatusLoader = RS_WaitRequest THEN
				sRunData.eCmdLoader := RCLo_GivePart;
				sRunData.TDataTable.iGiveTakeLayeringPosition := sRunData.TDataLoader.iLayringPos;
				sRunData.TDataTable.iGiveTakeLayeringOffsetPosition := sRunData.TDataLoader.iLayringOffsetPos;
				sRunData.eCmdTable := RCT_TakePart;
				eManagerStep := SP_RunStp44;
			END_IF
		SP_RunStp44:
			IF sRunData.sStatusLoader = RS_WaitRequest AND  sRunData.sStatusTable = RS_WaitRequest  THEN
				IF sCmd.TPickPlace.Activate THEN
					eManagerStep := SP_RunStp30;(* Skip *)
				ELSE
					eManagerStep := SP_RunStp1;(* End *)
				END_IF
			END_IF
		SP_RunStp50:
			IF sRunData.sStatusPearling = RS_WaitRequest THEN
				bDoChangeTool := FALSE;
				eManagerStep := SP_RunStp1;
			END_IF
	END_CASE
END_IF

END_FUNCTION_BLOCK

// ---- POUs/Manager/ManagerRun.TcPOU

FUNCTION_BLOCK ManagerRun
VAR_INPUT
	bPurging					: BOOL;
	bFirstCycle					: BOOL;
	bNewJob						: BOOL;
	sConfigFileData				: TConfigFileData;
	sProdLot					: TProductionLot;
	bLayeringWithTwoParts		: BOOL;
	bSimPearling				: BOOL;
	bDisableCleanAfterPearling	: BOOL;
END_VAR
VAR_OUTPUT
	bRecipeIsFinish				: BOOL;
	bConfigError				: BOOL;
END_VAR
VAR_IN_OUT
	sRunData					: TRunData;
	sProductionCmd				: TProductionCmd;
END_VAR
VAR
	i(*,j,k*)					: INT;
	iPartOnProcess				: INT;
	iPartOnLoader				: INT;
	iPartOnTurnOver				: INT;
	iPartOnTable				: INT;

	iGoodPartOnProcess			: INT;
	iGoodPartOnLoader			: INT;
	iGoodPartOnTurnOver			: INT;
	iGoodPartOnTable			: INT;


	bNeedNewPart				: BOOL;
	bLayering1IsSous			: BOOL;
	bPearlsOnBothSide			: BOOL;
	bPearlsOnSideSus			: BOOL;
	bPearlsOnSideSous			: BOOL;
(*	bDoNothing					: BOOL;*)
	bUseTurnOver				: BOOL;
	ePearlingTableSide			: TTableSide;
	eWorkingTableSide			: TTableSide;
	iLayeringPos				: INT;
	iLayeringOffsetPos			: INT;
	iHead						: INT;
	iSide						: INT;
(*	iPartSide					: INT;*)
	iMaxLayeringOffsetPos		: INT;
	eManagerStep				: TModuleSteps;
	eRestartStep				: TModuleSteps;
	eRestartLoaderStep			: TModuleSteps;
	bReadyForPearling			: BOOL;
(*	bReadyForTurn				: BOOL;
	bRecoveryFinish				: BOOL;*)
	bTableIsClean				: BOOL;
	bPearlingFinishOnTableSide	: BOOL;
	iRunLayering				: INT;
	iRunLayeringOffset			: INT;
	iStep						: INT;
	bLastPart					: BOOL;
	bTablePos2NeedPart			: BOOL;
END_VAR
(* Only for testing *)
VAR PERSISTENT
	bTestLift1ToLift2			: BOOL;
	bTestLift1ToTableRotationToLift2 : BOOL;
	bTestLift1ToTableToLift2	: BOOL;
END_VAR

sRunData.eCmdTurnOver := RCTO_None;
sRunData.eCmdTable := RCT_None;
sRunData.eCmdLoader := RCLo_None;
sRunData.eCmdPearling := RCP_None;

IF bFirstCycle THEN
	(* Put here variable that need to be reset between each start of the run *)
	eManagerStep := SP_InitStp1;
	sProductionCmd.TRequestSample.Activate := FALSE;
	sProductionCmd.TAutoSampling.iPeriodCnt := 0;
	sProductionCmd.TAutoSampling.iBatchCnt := 0;
END_IF

IF bNewJob THEN
	bReadyForPearling := FALSE;
	eWorkingTableSide := TS_A;
	eRestartStep := SP_RunStp1;
	eRestartLoaderStep := SP_RunStp1;
	sProductionCmd.TAutoSampling.iPeriodCnt := 0;
	sProductionCmd.TAutoSampling.iBatchCnt := 0;
END_IF

IF NOT bUseASOption THEN
	 sProductionCmd.TAutoSampling.bEnable := FALSE;
END_IF

IF NOT sProductionCmd.TAutoSampling.bEnable THEN
	sProductionCmd.TAutoSampling.iPeriodCnt := 0;
	sProductionCmd.TAutoSampling.iBatchCnt := 0;
END_IF

sProductionCmd.TRequestSample.Enable := NOT sProductionCmd.TAutoSampling.bEnable AND NOT sProductionCmd.TRequestSample.Activate;

(* Compute some data *)

IF bLayeringWithTwoParts THEN
	iMaxLayeringOffsetPos := 1;
ELSE
	iMaxLayeringOffsetPos := 0;
END_IF

bPearlsOnSideSus := sConfigFileData.asPearlingData[PS_SUS].THead[PH_Left].nNbOfPearls>0 OR sConfigFileData.asPearlingData[PS_SUS].THead[PH_Right].nNbOfPearls>0 ;
bPearlsOnSideSous := sConfigFileData.asPearlingData[PS_SOUS].THead[PH_Left].nNbOfPearls>0 OR sConfigFileData.asPearlingData[PS_SOUS].THead[PH_Right].nNbOfPearls>0 ;
bPearlsOnBothSide := bPearlsOnSideSus AND bPearlsOnSideSous;
IF sConfigFileData.bParallelProduction THEN
	bLayering1IsSous := FALSE;
ELSE
	bLayering1IsSous := TRUE;
END_IF
bUseTurnOver := bPearlsOnSideSous AND bLayering1IsSous;

iPartOnLoader := 0;
iGoodPartOnLoader := 0;
//IF sRunData.sStatusLoader = RS_WaitRequest THEN
	FOR iHead:= LH_Head1 TO LH_Head2 DO
		IF sRunData.TDataLoader.aTPartData[iHead].bPartPresent THEN
			iPartOnLoader := iPartOnLoader + 1;
			IF NOT sRunData.TDataLoader.aTPartData[iHead].bToReject THEN
				iGoodPartOnLoader := iGoodPartOnLoader + 1;
			END_IF
		END_IF
	END_FOR
//END_IF

iPartOnTable := 0;
iGoodPartOnTable := 0;
//IF sRunData.sStatusTable = RS_WaitRequest THEN
	FOR iLayeringPos:= 0 TO 1 DO
		FOR iLayeringOffsetPos:= 0 TO iMaxLayeringOffsetPos DO
			FOR iSide:= TS_A TO TS_B DO
				IF sRunData.TDataTable.aTPartData[iLayeringPos,iLayeringOffsetPos,iSide].bPartPresent THEN
					iPartOnTable := iPartOnTable + 1;
					IF NOT sRunData.TDataTable.aTPartData[iLayeringPos,iLayeringOffsetPos,iSide].bToReject THEN
						iGoodPartOnTable := iGoodPartOnTable + 1;
					END_IF
				END_IF
			END_FOR
		END_FOR
	END_FOR
//END_IF

iPartOnTurnOver := 0;
iGoodPartOnTurnOver := 0;
//IF sRunData.sStatusTurnOver = RS_WaitRequest AND bUseTurnOver THEN
	FOR i:= TO_Arm TO TO_Fix DO
		IF sRunData.TDataTurnOver.aTPartData[i].bPartPresent THEN
			iPartOnTurnOver := iPartOnTurnOver + 1;
			IF NOT sRunData.TDataTurnOver.aTPartData[i].bToReject THEN
				iGoodPartOnTurnOver := iGoodPartOnTurnOver + 1;
			END_IF
		END_IF
	END_FOR
//END_IF

iPartOnProcess := iPartOnLoader + iPartOnTurnOver + iPartOnTable;
iGoodPartOnProcess := iGoodPartOnLoader + iGoodPartOnTurnOver + iGoodPartOnTable;
bNeedNewPart := FALSE;
IF C_PROD_MODE_GOOD_PART THEN
	IF sProdLot.dGoodQty + INT_TO_DWORD(iGoodPartOnProcess) < sProdLot.dLotQty THEN
		bNeedNewPart := TRUE;
	END_IF
ELSE
	IF sProdLot.dLoadedQty < sProdLot.dLotQty THEN
		bNeedNewPart := TRUE;
	END_IF
END_IF
IF bPurging THEN
	bNeedNewPart := FALSE;
END_IF

IF sRunData.TDataTable.eTableSide = TS_A THEN
	ePearlingTableSide := TS_B;
ELSE
	ePearlingTableSide := TS_A;
END_IF

(* Part status updated *)

IF bTestLift1ToLift2 THEN
	CASE eManagerStep OF
		SP_InitStp1:	(*Recovery, Drop plate if we have one*)
			IF sRunData.TDataLoader.bPlatePresent THEN
				sRunData.eCmdLoader := RCLo_SwitchPlate;
				eManagerStep := SP_InitStp2;
			ELSE
				eManagerStep := SP_InitStp3;
			END_IF
		SP_InitStp2: (* Switch plate done *)
			IF sRunData.sStatusLoader = RS_WaitRequest THEN
				eManagerStep := SP_InitStp3;
			END_IF
		SP_InitStp3: (* Do we need a table turn ? *)
			IF  sRunData.TDataTable.eTableSide <>  eWorkingTableSide THEN
				sRunData.eCmdTable := RCT_Turn;
				eManagerStep := SP_InitStp4;
			ELSE
				eManagerStep := SP_InitStp5;
			END_IF
		SP_InitStp4:
				IF sRunData.sStatusTable = RS_WaitRequest THEN
					eManagerStep := SP_InitStp5;
				END_IF
		SP_InitStp5:
			IF sRunData.TDataLoader.aTPartData[LH_Head1].bPartPresent OR sRunData.TDataLoader.aTPartData[LH_Head2].bPartPresent THEN
				eManagerStep := eRestartLoaderStep;
			ELSE
				eManagerStep := eRestartStep;
			END_IF
(* Running Step *)
		SP_RunStp1:
			eRestartStep := SP_RunStp1;
			eRestartLoaderStep := SP_RunStp1;
			eManagerStep := SP_RunStp10;
		SP_RunStp10:
			(* Take part on head 1 from loader *)
			IF sRunData.TDataLoader.aTPartData[LH_Head1].bPartPresent THEN
				eManagerStep := SP_RunStp20;
			ELSE
				sRunData.TDataLoader.eModule := LMP_Lift1;
				sRunData.TDataLoader.eTaker := LH_Head1;
				sRunData.eCmdLoader := RCLo_PrepareTakePart;
				eManagerStep := SP_RunStp11;
			END_IF
		SP_RunStp11:
			IF sRunData.sStatusLoader = RS_WaitRequest THEN
				sRunData.eCmdLoader := RCLo_TakePart;
				eManagerStep := SP_RunStp12;
			END_IF
		SP_RunStp12:
			IF sRunData.sStatusLoader = RS_WaitRequest THEN
				eManagerStep := SP_RunStp20;
			END_IF
		SP_RunStp20:
			(* Take part on head 2 from loader *)
			IF sRunData.TDataLoader.aTPartData[LH_Head2].bPartPresent THEN
				eManagerStep := SP_RunStp30;
			ELSE
				sRunData.TDataLoader.eModule := LMP_Lift1;
				sRunData.TDataLoader.eTaker := LH_Head2;
				sRunData.eCmdLoader := RCLo_PrepareTakePart;
				eManagerStep := SP_RunStp21;
			END_IF
		SP_RunStp21:
				IF sRunData.sStatusLoader = RS_WaitRequest THEN
				sRunData.eCmdLoader := RCLo_TakePart;
				eManagerStep := SP_RunStp22;
			END_IF
		SP_RunStp22:
			IF sRunData.sStatusLoader = RS_WaitRequest THEN
				eManagerStep := SP_RunStp30;
			END_IF
		SP_RunStp30:
			(* Drop part from head 1 to unloader *)
			sRunData.TDataLoader.eModule := LMP_Lift2;
			sRunData.TDataLoader.eTaker := LH_Head1;
			sRunData.eCmdLoader := RCLo_PrepareDropPart;
			eManagerStep := SP_RunStp31;
		SP_RunStp31:
			IF sRunData.sStatusLoader = RS_WaitRequest THEN
				sRunData.eCmdLoader := RCLo_GivePart;
				eManagerStep := SP_RunStp32;
			END_IF
		SP_RunStp32:
			IF sRunData.sStatusLoader = RS_WaitRequest THEN
				eManagerStep := SP_RunStp40;
			END_IF
		SP_RunStp40:
			(* Drop part from head 2 to unloader *)
			sRunData.TDataLoader.eModule := LMP_Lift2;
			sRunData.TDataLoader.eTaker := LH_Head2;
			sRunData.eCmdLoader := RCLo_PrepareDropPart;
			eManagerStep := SP_RunStp41;
		SP_RunStp41:
			IF sRunData.sStatusLoader = RS_WaitRequest THEN
				sRunData.eCmdLoader := RCLo_GivePart;
				eManagerStep := SP_RunStp42;
			END_IF
		SP_RunStp42:
			IF sRunData.sStatusLoader = RS_WaitRequest THEN
				eManagerStep := SP_RunStp1;
			END_IF
	END_CASE

// HFO -->
ELSIF bTestLift1ToTableRotationToLift2 THEN
	CASE eManagerStep OF
		SP_InitStp1:	(*Recovery, Drop plate if we have one*)
			bTableIsClean := FALSE;
			IF sRunData.TDataLoader.bPlatePresent THEN
				sRunData.eCmdLoader := RCLo_SwitchPlate;
				eManagerStep := SP_InitStp2;
			ELSE
				eManagerStep := SP_InitStp3;
			END_IF
		SP_InitStp2: (* Switch plate done *)
			IF sRunData.sStatusLoader = RS_WaitRequest THEN
				eManagerStep := SP_InitStp3;
			END_IF
		SP_InitStp3: (* Do we need a table turn ? *)
			IF  sRunData.TDataTable.eTableSide <>  eWorkingTableSide THEN
				sRunData.eCmdTable := RCT_Turn;
				eManagerStep := SP_InitStp4;
			ELSE
				eManagerStep := SP_InitStp5;
			END_IF
		SP_InitStp4:
				IF sRunData.sStatusTable = RS_WaitRequest THEN
					eManagerStep := SP_InitStp5;
				END_IF
		SP_InitStp5:
			IF sRunData.TDataLoader.aTPartData[LH_Head1].bPartPresent THEN
				eManagerStep := eRestartLoaderStep;
			ELSE
				eManagerStep := eRestartStep;
			END_IF
(* Running Step *)
		SP_RunStp1:
			sRunData.TDataLoader.iLayringOffsetPos := 0;
			sRunData.TDataTable.iGiveTakeLayeringOffsetPosition := sRunData.TDataLoader.iLayringOffsetPos;
			eRestartStep := SP_RunStp1;
			eRestartLoaderStep := SP_RunStp1;
			// Check if parts can be taken on table
			IF sRunData.TDataTable.aTPartData[0,0,sRunData.TDataTable.eTableSide].bPartPresent
					AND NOT sRunData.TDataLoader.aTPartData[0].bPartPresent THEN
				// Take the part on table with head1
				bTableIsClean := FALSE;
				sRunData.TDataLoader.eModule := LMP_Table;
				sRunData.TDataLoader.eTaker := LH_Head1;
				sRunData.TDataLoader.iLayringPos := 0;
				eManagerStep := SP_RunStp100;
			ELSIF sRunData.TDataTable.aTPartData[1,0,sRunData.TDataTable.eTableSide].bPartPresent
					AND NOT sRunData.TDataLoader.aTPartData[1].bPartPresent THEN
				// Take the part on table with head2
				bTableIsClean := FALSE;
				sRunData.TDataLoader.eModule := LMP_Table;
				sRunData.TDataLoader.eTaker := LH_Head2;
				sRunData.TDataLoader.iLayringPos := 1;
				eManagerStep := SP_RunStp100;
			ELSIF NOT sRunData.TDataLoader.aTPartData[0].bPartPresent 
					AND NOT sRunData.TDataLoader.aTPartData[1].bPartPresent THEN
				// Move loader to safe for cleaning and reload
				sRunData.eCmdLoader := RCLo_MoveToSafe;
				eManagerStep := SP_RunStp50;
			ELSE
				// Move loader to safe and drop part
				sRunData.eCmdLoader := RCLo_MoveToSafe;
				eManagerStep := SP_RunStp2;
			END_IF
		SP_RunStp2: // Drop parts and check table
			IF sRunData.sStatusLoader = RS_WaitRequest THEN
				// Check if table can be cleaned
				IF sRunData.sStatusTable = RS_WaitRequest
						AND NOT sRunData.TDataTable.aTPartData[0,0,sRunData.TDataTable.eTableSide].bPartPresent
						AND NOT sRunData.TDataTable.aTPartData[1,0,sRunData.TDataTable.eTableSide].bPartPresent 
						AND NOT bTableIsClean THEN
					// Clean the table
					sRunData.eCmdTable := RCT_Clean;
				END_IF
				// Check if part must be dropped
				IF sRunData.TDataLoader.aTPartData[0].bPartPresent THEN
					// Drop part on head 1
					sRunData.TDataLoader.eTaker := LH_Head1;
					eManagerStep := SP_RunStp200;
				ELSIF sRunData.TDataLoader.aTPartData[1].bPartPresent THEN
					// Drop part on head 2
					sRunData.TDataLoader.eTaker := LH_Head2;
					eManagerStep := SP_RunStp200;
				ELSIF sRunData.sStatusTable = RS_WaitRequest THEN
					// No more parts on head and table is clean
					bTableIsClean := TRUE;
					eManagerStep := SP_RunStp1;
				END_IF
			END_IF

		SP_RunStp50: // Do cleaning and reload from lift
			eRestartStep := SP_RunStp50;
			eRestartLoaderStep := SP_RunStp50;
			IF sRunData.sStatusLoader = RS_WaitRequest THEN
				// Check if table can be cleaned
				IF sRunData.sStatusTable = RS_WaitRequest AND NOT bTableIsClean THEN
					// Clean the table
					sRunData.eCmdTable := RCT_Clean;
				END_IF
				IF bNeedNewPart THEN
					IF NOT sRunData.TDataLoader.aTPartData[0].bPartPresent AND NOT bTablePos2NeedPart THEN
						sRunData.TDataLoader.eModule := LMP_Lift1;
						sRunData.TDataLoader.eTaker := LH_Head1;
						sRunData.eCmdLoader := RCLo_PrepareTakePart;
						eManagerStep := SP_RunStp55;
					ELSIF NOT sRunData.TDataLoader.aTPartData[1].bPartPresent THEN
						sRunData.TDataLoader.eModule := LMP_Lift1;
						sRunData.TDataLoader.eTaker := LH_Head2;
						sRunData.eCmdLoader := RCLo_PrepareTakePart;
						eManagerStep := SP_RunStp55;
					ELSIF sRunData.sStatusTable = RS_WaitRequest THEN
						bTableIsClean := TRUE;
						eManagerStep := SP_RunStp70;
					END_IF	
				ELSE
					eManagerStep := SP_RunStp80;
					// eManagerStep := SP_RunStp160; 	// purging
				END_IF
			END_IF				
		SP_RunStp55:
			IF sRunData.sStatusLoader = RS_WaitRequest THEN
				sRunData.eCmdLoader := RCLo_TakePart;
				eManagerStep := SP_RunStp60;
			END_IF
		SP_RunStp60:
			IF sRunData.sStatusLoader = RS_WaitRequest 
					AND sRunData.sStatusTable = RS_WaitRequest THEN
				bTableIsClean := TRUE;
				eManagerStep := SP_RunStp50;
			END_IF
		SP_RunStp70: (* Drop part on layering *)
			IF sRunData.sStatusTable = RS_WaitRequest THEN
				eRestartStep := SP_RunStp70;
				eRestartLoaderStep := SP_RunStp70;
				IF sRunData.TDataLoader.aTPartData[0].bPartPresent THEN
					IF sRunData.TDataLoader.aTPartData[0].bToReject THEN
						sRunData.TDataLoader.eModule := LMP_Reject;
						sRunData.TDataLoader.eTaker := LH_Head1;
						sRunData.eCmdLoader := RCLo_PrepareDropPart;
						eManagerStep := SP_RunStp150;
					ELSE
						sRunData.TDataLoader.eModule := LMP_Table;
						sRunData.TDataLoader.eTaker := LH_Head1;
						sRunData.TDataLoader.iLayringPos := 0;
						sRunData.eCmdLoader := RCLo_PrepareDropPart;
						eManagerStep := SP_RunStp75;
					END_IF
				ELSIF sRunData.TDataLoader.aTPartData[1].bPartPresent THEN
					IF sRunData.TDataLoader.aTPartData[1].bToReject THEN
						sRunData.TDataLoader.eModule := LMP_Reject;
						sRunData.TDataLoader.eTaker := LH_Head2;
						sRunData.eCmdLoader := RCLo_PrepareDropPart;
						bTablePos2NeedPart := TRUE;
						eManagerStep := SP_RunStp150;
					ELSE
						sRunData.TDataLoader.eModule := LMP_Table;
						sRunData.TDataLoader.eTaker := LH_Head2;
						sRunData.TDataLoader.iLayringPos := 1;
						sRunData.eCmdLoader := RCLo_PrepareDropPart;
						bTablePos2NeedPart := FALSE;
						eManagerStep := SP_RunStp75;
					END_IF
				ELSE
					// Loading finished, turn table
					eManagerStep := SP_RunStp80;
				END_IF
			END_IF
		SP_RunStp75:
			IF sRunData.sStatusLoader = RS_WaitRequest THEN
				sRunData.TDataTable.iGiveTakeLayeringPosition := sRunData.TDataLoader.iLayringPos;
				sRunData.eCmdLoader := RCLo_GivePart;
				sRunData.eCmdTable := RCT_TakePart;
				eManagerStep := SP_RunStp77;
			END_IF
		SP_RunStp77:
			IF sRunData.sStatusLoader = RS_WaitRequest AND  sRunData.sStatusTable = RS_WaitRequest  THEN
				eManagerStep := SP_RunStp70;
			END_IF		
		SP_RunStp80:
			IF sRunData.sStatusLoader = RS_WaitRequest AND  sRunData.sStatusTable = RS_WaitRequest  THEN
				sRunData.eCmdLoader := RCLo_MoveToSafe;
				eManagerStep := SP_RunStp85;
			END_IF		
		SP_RunStp85:
			IF sRunData.sStatusLoader = RS_WaitRequest THEN
				(* Pearling finish *)
				eManagerStep := SP_RunStp90;
			END_IF
		SP_RunStp90:
			eRestartStep := SP_RunStp96;
			eRestartLoaderStep := SP_RunStp93;
			sRunData.eCmdTable := RCT_Turn;
			eWorkingTableSide := ePearlingTableSide;
			eManagerStep := SP_RunStp93;
		SP_RunStp93: (*Turning Table *)
			IF sRunData.sStatusTable = RS_ProcessRequest2 THEN
				IF iPartOnProcess = 0 AND NOT bNeedNewPart THEN
					eManagerStep := SP_RunStp300;
				ELSE
					bReadyForPearling := TRUE;
					eManagerStep := SP_RunStp96;
				END_IF
			END_IF
		SP_RunStp96: (*Cleaning Table *)
			IF sRunData.sStatusTable = RS_WaitRequest  AND  sRunData.sStatusLoader = RS_WaitRequest  THEN
				bTableIsClean := TRUE;
				eManagerStep := SP_RunStp1;
			END_IF
		SP_RunStp100: (* Unloading part on layering *)
			eRestartStep := SP_RunStp100;
			eRestartLoaderStep := SP_RunStp100;
			sRunData.TDataLoader.eModule := LMP_Table;
			sRunData.eCmdLoader := RCLo_PrepareTakePart;
			eManagerStep := SP_RunStp105;
		SP_RunStp105:
			IF sRunData.sStatusLoader = RS_WaitRequest THEN
				sRunData.eCmdLoader := RCLo_TakePart;
				sRunData.TDataTable.iGiveTakeLayeringPosition := sRunData.TDataLoader.iLayringPos;
				sRunData.TDataTable.iGiveTakeLayeringOffsetPosition := sRunData.TDataLoader.iLayringOffsetPos;
				sRunData.eCmdTable := RCT_GivePart;
				eManagerStep := SP_RunStp110;
			END_IF
		SP_RunStp110:
			IF sRunData.sStatusLoader = RS_WaitRequest AND  sRunData.sStatusTable = RS_WaitRequest  THEN
				eManagerStep := SP_RunStp1;
			END_IF
		SP_RunStp150: // Give bad part to the reject
			IF sRunData.sStatusLoader = RS_WaitRequest THEN
				sRunData.eCmdLoader := RCLo_GivePart;
				eManagerStep := SP_RunStp151;
			END_IF
		SP_RunStp151:
			IF sRunData.sStatusLoader = RS_WaitRequest THEN
				eManagerStep := SP_RunStp50;
			END_IF
		SP_RunStp160: // TODO : (HFO) // Steps for purging 
			IF sRunData.sStatusLoader = RS_WaitRequest AND  sRunData.sStatusTable = RS_WaitRequest  THEN
				sRunData.eCmdLoader := RCLo_MoveToSafe;
				//eManagerStep := SP_RunStp85;
			END_IF		
		SP_RunStp200:
			IF sRunData.sStatusLoader = RS_WaitRequest THEN
				IF sRunData.TDataLoader.aTPartData[LH_Head1].bToReject THEN
					sRunData.TDataLoader.eModule := LMP_Reject;
				ELSIF sProductionCmd.TRequestSample.Activate THEN
					sRunData.TDataLoader.eModule := LMP_Sample;
					sProductionCmd.TRequestSample.Activate := FALSE;
				ELSE
					sProductionCmd.TAutoSampling.iPeriodCnt := sProductionCmd.TAutoSampling.iPeriodCnt + 1;
					IF sProductionCmd.TAutoSampling.bEnable AND (sProductionCmd.TAutoSampling.iPeriodCnt >= (sProductionCmd.TAutoSampling.iPeriod - sProductionCmd.TAutoSampling.iBatchSize)) THEN
						sRunData.TDataLoader.eModule := LMP_Sample;
						sProductionCmd.TAutoSampling.iBatchCnt := sProductionCmd.TAutoSampling.iBatchCnt + 1;
						IF sProductionCmd.TAutoSampling.iBatchCnt >= sProductionCmd.TAutoSampling.iBatchSize THEN
							sProductionCmd.TAutoSampling.iBatchCnt := 0;
							sProductionCmd.TAutoSampling.iPeriodCnt := 0;
						END_IF
					ELSE
						sRunData.TDataLoader.eModule := LMP_Lift2;
					END_IF
				END_IF
				sRunData.eCmdLoader := RCLo_PrepareDropPart;
				eManagerStep := SP_RunStp205;
			END_IF
		SP_RunStp205:
			IF sRunData.sStatusLoader = RS_WaitRequest THEN
				sRunData.eCmdLoader := RCLo_GivePart;
				eManagerStep := SP_RunStp210;
			END_IF
		SP_RunStp210:
			IF sRunData.sStatusLoader = RS_WaitRequest THEN
				bTableIsClean := TRUE;
				eManagerStep := SP_RunStp2;
			END_IF
		SP_RunStp300: (*End of recipe *)
			bReadyForPearling := FALSE;
			sRunData.eCmdLoader := RCLo_EndOfRecipe;
			eManagerStep := SP_RunStp305;
		SP_RunStp305: (*Loader in safe and lift in unload position *)
			IF sRunData.sStatusLoader = RS_WaitRequest  AND sRunData.sStatusPearling = RS_WaitRequest AND sRunData.sStatusTable = RS_WaitRequest THEN
				eManagerStep := SP_RunStp0;
			END_IF
	END_CASE
// HFO <--
	
ELSIF bTestLift1ToTableToLift2 THEN
	CASE eManagerStep OF
		SP_InitStp1:	(*Recovery, Drop plate if we have one*)
			IF sRunData.TDataLoader.bPlatePresent THEN
				sRunData.eCmdLoader := RCLo_SwitchPlate;
				eManagerStep := SP_InitStp2;
			ELSE
				eManagerStep := SP_InitStp3;
			END_IF
		SP_InitStp2: (* Switch plate done *)
			IF sRunData.sStatusLoader = RS_WaitRequest THEN
				eManagerStep := SP_InitStp3;
			END_IF
		SP_InitStp3: (* Do we need a table turn ? *)
			IF  sRunData.TDataTable.eTableSide <>  eWorkingTableSide THEN
				sRunData.eCmdTable := RCT_Turn;
				eManagerStep := SP_InitStp4;
			ELSE
				eManagerStep := SP_InitStp5;
			END_IF
		SP_InitStp4:
				IF sRunData.sStatusTable = RS_WaitRequest THEN
					eManagerStep := SP_InitStp5;
				END_IF
		SP_InitStp5:
			IF sRunData.TDataLoader.aTPartData[LH_Head1].bPartPresent OR sRunData.TDataLoader.aTPartData[LH_Head2].bPartPresent THEN
				eManagerStep := eRestartLoaderStep;
			ELSE
				eManagerStep := eRestartStep;
			END_IF
(* Running Step *)
		SP_RunStp1:
			eRestartStep := SP_RunStp1;
			eRestartLoaderStep := SP_RunStp1;
			eManagerStep := SP_RunStp2;
		SP_RunStp2:
			(* Check if part present on table A/C*)
			IF sRunData.TDataTable.aTPartData[0,0,sRunData.TDataTable.eTableSide].bPartPresent THEN
				sRunData.TDataLoader.iLayringPos := 0;
				eManagerStep := SP_RunStp40;
			(* Check if part present on table B/D*)
			ELSIF sRunData.TDataTable.aTPartData[1,0,sRunData.TDataTable.eTableSide].bPartPresent THEN
				sRunData.TDataLoader.iLayringPos := 1;
				eManagerStep := SP_RunStp40;
			ELSE
				IF NOT sRunData.TDataLoader.aTPartData[LH_Head1].bPartPresent THEN
					eManagerStep := SP_RunStp30;
				ELSE
					eManagerStep := SP_RunStp60;
				END_IF
			END_IF
		SP_RunStp10:
			(* Take part on head 1 from loader *)
			IF sRunData.TDataLoader.aTPartData[LH_Head1].bPartPresent THEN
				eManagerStep := SP_RunStp20;
			ELSE
				sRunData.TDataLoader.eModule := LMP_Lift1;
				sRunData.TDataLoader.eTaker := LH_Head1;
				sRunData.eCmdLoader := RCLo_PrepareTakePart;
				eManagerStep := SP_RunStp11;
			END_IF
		SP_RunStp11:
			IF sRunData.sStatusLoader = RS_WaitRequest THEN
				sRunData.eCmdLoader := RCLo_TakePart;
				eManagerStep := SP_RunStp12;
			END_IF
		SP_RunStp12:
			IF sRunData.sStatusLoader = RS_WaitRequest THEN
				eManagerStep := SP_RunStp20;
			END_IF
		SP_RunStp20:
			(* Drop part on head 1 on table *)
			sRunData.TDataLoader.eModule := LMP_Table;
			sRunData.TDataLoader.eTaker := LH_Head1;
			sRunData.TDataLoader.iLayringPos := 1;
			sRunData.TDataLoader.iLayringOffsetPos := 0;
			sRunData.eCmdLoader := RCLo_PrepareDropPart;
			eManagerStep := SP_RunStp21;
		SP_RunStp21:
			IF sRunData.sStatusLoader = RS_WaitRequest THEN
				sRunData.eCmdLoader := RCLo_GivePart;
				sRunData.TDataTable.iGiveTakeLayeringPosition := sRunData.TDataLoader.iLayringPos;
				sRunData.TDataTable.iGiveTakeLayeringOffsetPosition := sRunData.TDataLoader.iLayringOffsetPos;
				sRunData.eCmdTable := RCT_TakePart;
				eManagerStep := SP_RunStp22;
			END_IF
		SP_RunStp22:
			IF sRunData.sStatusLoader = RS_WaitRequest AND sRunData.sStatusTable = RS_WaitRequest THEN
				IF NOT sRunData.TDataLoader.aTPartData[LH_Head1].bPartPresent THEN
					eManagerStep := SP_RunStp30;
				END_IF
			END_IF
		SP_RunStp30:
			(* Take part on head 1 from loader *)
			sRunData.TDataLoader.eModule := LMP_Lift1;
			sRunData.TDataLoader.eTaker := LH_Head1;
			eManagerStep := SP_RunStp31;
			IF NOT sRunData.TDataTable.aTPartData[0,0,sRunData.TDataTable.eTableSide].bPartPresent THEN
				sRunData.eCmdLoader := RCLo_PrepareTakePart;
				sRunData.TDataLoader.iLayringPos := 0;
			ELSIF NOT sRunData.TDataTable.aTPartData[1,0,sRunData.TDataTable.eTableSide].bPartPresent THEN
				sRunData.eCmdLoader := RCLo_PrepareTakePart;
				sRunData.TDataLoader.iLayringPos := 1;
			ELSE
				eManagerStep := SP_RunStp2;
			END_IF
		SP_RunStp31:
				IF sRunData.sStatusLoader = RS_WaitRequest THEN
				sRunData.eCmdLoader := RCLo_TakePart;
				eManagerStep := SP_RunStp32;
			END_IF
		SP_RunStp32:
			IF sRunData.sStatusLoader = RS_WaitRequest THEN
				eManagerStep := SP_RunStp50;
			END_IF
		SP_RunStp40:
			(* Take part on head 1 from table *)
			sRunData.TDataLoader.eModule := LMP_Table;
			sRunData.TDataLoader.eTaker := LH_Head1;
			sRunData.TDataLoader.iLayringOffsetPos := 0;
			sRunData.eCmdLoader := RCLo_PrepareTakePart;
			eManagerStep := SP_RunStp41;
		SP_RunStp41:
			IF sRunData.sStatusLoader = RS_WaitRequest THEN
				sRunData.eCmdLoader := RCLo_TakePart;
				sRunData.TDataTable.iGiveTakeLayeringPosition := sRunData.TDataLoader.iLayringPos;
				sRunData.TDataTable.iGiveTakeLayeringOffsetPosition := sRunData.TDataLoader.iLayringOffsetPos;
				sRunData.eCmdTable := RCT_GivePart;
				eManagerStep := SP_RunStp42;
			END_IF
		SP_RunStp42:
			IF sRunData.sStatusLoader = RS_WaitRequest AND  sRunData.sStatusTable = RS_WaitRequest  THEN
				eManagerStep := SP_RunStp60;
			END_IF
		SP_RunStp50:
			(* Drop part on head 1 on table *)
			sRunData.TDataLoader.eModule := LMP_Table;
			sRunData.TDataLoader.eTaker := LH_Head1;
			sRunData.TDataLoader.iLayringOffsetPos := 0;
			sRunData.eCmdLoader := RCLo_PrepareDropPart;
			eManagerStep := SP_RunStp51;
		SP_RunStp51:
			IF sRunData.sStatusLoader = RS_WaitRequest THEN
				sRunData.eCmdLoader := RCLo_GivePart;
				sRunData.TDataTable.iGiveTakeLayeringPosition := sRunData.TDataLoader.iLayringPos;
				sRunData.TDataTable.iGiveTakeLayeringOffsetPosition := sRunData.TDataLoader.iLayringOffsetPos;
				sRunData.eCmdTable := RCT_TakePart;
				eManagerStep := SP_RunStp52;
			END_IF
		SP_RunStp52:
			IF sRunData.sStatusLoader = RS_WaitRequest AND sRunData.sStatusTable = RS_WaitRequest THEN
				IF NOT sRunData.TDataLoader.aTPartData[LH_Head1].bPartPresent THEN
					eManagerStep := SP_RunStp30;
				END_IF
			END_IF
		SP_RunStp60:
			(* Drop part from head 1 to unloader *)
			sRunData.TDataLoader.eModule := LMP_Lift2;
			sRunData.TDataLoader.eTaker := LH_Head1;
			sRunData.eCmdLoader := RCLo_PrepareDropPart;
			eManagerStep := SP_RunStp61;
		SP_RunStp61:
			IF sRunData.sStatusLoader = RS_WaitRequest THEN
				sRunData.eCmdLoader := RCLo_GivePart;
				eManagerStep := SP_RunStp62;
			END_IF
		SP_RunStp62:
			IF sRunData.sStatusLoader = RS_WaitRequest THEN
				eManagerStep := SP_RunStp2;
			END_IF
	END_CASE
ELSIF NOT sConfigFileData.bParallelProduction AND NOT bLayeringWithTwoParts THEN
	IF sRunData.sStatusPearling <> RS_WaitRequest THEN
		bPearlingFinishOnTableSide := FALSE;
	ELSE
		bPearlingFinishOnTableSide := TRUE;
		IF	(
				sRunData.TDataTable.aTPartData[0,0,ePearlingTableSide].bPartPresent AND
				NOT sRunData.TDataTable.aTPartData[0,0,ePearlingTableSide].abPearlingDone[PH_Left,PS_SUS] AND
				sConfigFileData.asPearlingData[PS_SUS].THead[PH_Left].nNbOfPearls > 0
			) OR (
				 sRunData.TDataTable.aTPartData[0,0,ePearlingTableSide].bPartPresent AND
				NOT sRunData.TDataTable.aTPartData[0,0,ePearlingTableSide].abPearlingDone[PH_Right,PS_SUS] AND
				sConfigFileData.asPearlingData[PS_SUS].THead[PH_Right].nNbOfPearls > 0
			) OR (
				sRunData.TDataTable.aTPartData[1,0,ePearlingTableSide].bPartPresent AND
				NOT sRunData.TDataTable.aTPartData[1,0,ePearlingTableSide].abPearlingDone[PH_Left,PS_SOUS] AND
				sConfigFileData.asPearlingData[PS_SOUS].THead[PH_Left].nNbOfPearls > 0
			) OR (
				sRunData.TDataTable.aTPartData[1,0,ePearlingTableSide].bPartPresent AND
				NOT sRunData.TDataTable.aTPartData[1,0,ePearlingTableSide].abPearlingDone[PH_Right,PS_SOUS] AND
				sConfigFileData.asPearlingData[PS_SOUS].THead[PH_Right].nNbOfPearls > 0
			) THEN
			bPearlingFinishOnTableSide := FALSE;
		END_IF
	END_IF
	CASE eManagerStep OF
		SP_InitStp1:	(*Recovery, Drop plate if we have one*)
			sRunData.eCmdPearling := RCP_CheckSharpen;
			bReadyForPearling := FALSE;
			bTableIsClean := FALSE;
			IF sRunData.TDataLoader.bPlatePresent THEN
				sRunData.eCmdLoader := RCLo_SwitchPlate;
				eManagerStep := SP_InitStp2;
			ELSE
				eManagerStep := SP_InitStp3;
			END_IF
		SP_InitStp2: (* Switch plate done *)
			IF sRunData.sStatusLoader = RS_WaitRequest THEN
				eManagerStep := SP_InitStp3;
			END_IF
		SP_InitStp3: (* Do we need a table turn ? *)
			IF  sRunData.TDataTable.eTableSide <>  eWorkingTableSide THEN
				sRunData.eCmdTable := RCT_Turn;
				eManagerStep := SP_InitStp4;
			ELSE
				eManagerStep := SP_InitStp5;
			END_IF
		SP_InitStp4:
				IF sRunData.sStatusTable = RS_WaitRequest THEN
					eManagerStep := SP_InitStp5;
				END_IF
		SP_InitStp5:
			bReadyForPearling := TRUE;
			IF sRunData.TDataLoader.aTPartData[LH_Head1].bPartPresent OR sRunData.TDataLoader.aTPartData[LH_Head2].bPartPresent THEN
				eManagerStep := eRestartLoaderStep;
			ELSE
				eManagerStep := eRestartStep;
			END_IF
	END_CASE
	IF bPearlsOnSideSus THEN
		CASE eManagerStep OF
(* Running Step *)
			SP_RunStp1:
				eRestartStep := SP_RunStp1;
				eRestartLoaderStep := SP_RunStp4;
				IF sRunData.TDataTable.aTPartData[1,0,sRunData.TDataTable.eTableSide].bPartPresent THEN
					bTableIsClean := FALSE;
					eManagerStep := SP_RunStp2;
				ELSE
					eManagerStep := SP_RunStp10; (* Skip *)
				END_IF
			SP_RunStp2: (* Unloading part on layering 1 *)
				sRunData.TDataLoader.eModule := LMP_Table;
				sRunData.TDataLoader.eTaker := LH_Head2;
				sRunData.TDataLoader.iLayringPos := 1;
				sRunData.TDataLoader.iLayringOffsetPos := 0;
				sRunData.eCmdLoader := RCLo_PrepareTakePart;
				eManagerStep := SP_RunStp3;
			SP_RunStp3:
				IF sRunData.sStatusLoader = RS_WaitRequest THEN
					sRunData.eCmdLoader := RCLo_TakePart;
					sRunData.TDataTable.iGiveTakeLayeringPosition := sRunData.TDataLoader.iLayringPos;
					sRunData.TDataTable.iGiveTakeLayeringOffsetPosition := sRunData.TDataLoader.iLayringOffsetPos;
					sRunData.eCmdTable := RCT_GivePart;
					eManagerStep := SP_RunStp4;
				END_IF
			SP_RunStp4:
				IF sRunData.sStatusLoader = RS_WaitRequest AND  sRunData.sStatusTable = RS_WaitRequest  THEN
					sRunData.eCmdLoader := RCLo_Cleaning;
					eManagerStep := SP_RunStp5;
				END_IF
			SP_RunStp5:
				IF sRunData.sStatusLoader = RS_WaitRequest  THEN
					IF sRunData.TDataLoader.aTPartData[LH_Head2].bToReject THEN
						sRunData.TDataLoader.eModule := LMP_Reject;
					ELSIF sProductionCmd.TRequestSample.Activate THEN
						sRunData.TDataLoader.eModule := LMP_Sample;
						sProductionCmd.TRequestSample.Activate := FALSE;
					ELSE
						sProductionCmd.TAutoSampling.iPeriodCnt := sProductionCmd.TAutoSampling.iPeriodCnt  + 1;
						IF sProductionCmd.TAutoSampling.bEnable AND (sProductionCmd.TAutoSampling.iPeriodCnt  >= (sProductionCmd.TAutoSampling.iPeriod-sProductionCmd.TAutoSampling.iBatchSize)) THEN
							sRunData.TDataLoader.eModule := LMP_Sample;
							sProductionCmd.TAutoSampling.iBatchCnt := sProductionCmd.TAutoSampling.iBatchCnt + 1;
							IF sProductionCmd.TAutoSampling.iBatchCnt >= sProductionCmd.TAutoSampling.iBatchSize THEN
								sProductionCmd.TAutoSampling.iBatchCnt := 0;
								sProductionCmd.TAutoSampling.iPeriodCnt := 0;
							END_IF
						ELSE
							sRunData.TDataLoader.eModule := LMP_Lift2;
						END_IF
					END_IF
					sRunData.eCmdLoader := RCLo_PrepareDropPart;
					eManagerStep := SP_RunStp6;
				END_IF
			SP_RunStp6:
				IF sRunData.sStatusLoader = RS_WaitRequest THEN
					sRunData.eCmdLoader := RCLo_GivePart;
					eManagerStep := SP_RunStp7;
				END_IF
			SP_RunStp7:
				IF sRunData.sStatusLoader = RS_WaitRequest THEN
					eManagerStep := SP_RunStp10;
				END_IF
			SP_RunStp10: (* Unloading part on layering 0 *)
				eRestartStep := SP_RunStp10;
				eRestartLoaderStep := SP_RunStp13;
				IF sRunData.TDataTable.aTPartData[0,0,sRunData.TDataTable.eTableSide].bPartPresent THEN
					bTableIsClean := FALSE;
					eManagerStep := SP_RunStp11;
				ELSE
					eManagerStep := SP_RunStp20;(* Skip *)
				END_IF
			SP_RunStp11:
				sRunData.TDataLoader.eModule := LMP_Table;
				sRunData.TDataLoader.eTaker := LH_Head1;
				sRunData.TDataLoader.iLayringPos := 0;
				sRunData.TDataLoader.iLayringOffsetPos := 0;
				sRunData.eCmdLoader := RCLo_PrepareTakePart;
				eManagerStep := SP_RunStp12;
			SP_RunStp12:
				IF sRunData.sStatusLoader = RS_WaitRequest THEN
					sRunData.eCmdLoader := RCLo_TakePart;
					sRunData.TDataTable.iGiveTakeLayeringPosition := sRunData.TDataLoader.iLayringPos;
					sRunData.TDataTable.iGiveTakeLayeringOffsetPosition := sRunData.TDataLoader.iLayringOffsetPos;
					sRunData.eCmdTable := RCT_GivePart;
					eManagerStep := SP_RunStp13;
				END_IF
			SP_RunStp13:
				IF sRunData.sStatusLoader = RS_WaitRequest AND  sRunData.sStatusTable = RS_WaitRequest  THEN
					IF bUseTurnOver THEN
						sRunData.eCmdLoader := RCLo_Cleaning;
						eManagerStep := SP_RunStp14;
					ELSE
						IF sRunData.TDataLoader.aTPartData[LH_Head2].bToReject THEN
							sRunData.TDataLoader.eModule := LMP_Reject;
						ELSIF sProductionCmd.TRequestSample.Activate THEN
							sRunData.TDataLoader.eModule := LMP_Sample;
							sProductionCmd.TRequestSample.Activate := FALSE;
						ELSE
							sProductionCmd.TAutoSampling.iPeriodCnt := sProductionCmd.TAutoSampling.iPeriodCnt + 1;
							IF sProductionCmd.TAutoSampling.bEnable AND (sProductionCmd.TAutoSampling.iPeriodCnt >= (sProductionCmd.TAutoSampling.iPeriod - sProductionCmd.TAutoSampling.iBatchSize)) THEN
								sRunData.TDataLoader.eModule := LMP_Sample;
								sProductionCmd.TAutoSampling.iBatchCnt := sProductionCmd.TAutoSampling.iBatchCnt + 1;
								IF sProductionCmd.TAutoSampling.iBatchCnt >= sProductionCmd.TAutoSampling.iBatchSize THEN
									sProductionCmd.TAutoSampling.iBatchCnt := 0;
									sProductionCmd.TAutoSampling.iPeriodCnt := 0;
								END_IF
							ELSE
								sRunData.TDataLoader.eModule := LMP_Lift2;
							END_IF
						END_IF
						sRunData.eCmdLoader := RCLo_PrepareDropPart;
						eManagerStep := SP_RunStp15;
					END_IF
				END_IF
			SP_RunStp14:
				IF sRunData.sStatusLoader = RS_WaitRequest THEN
					sRunData.eCmdLoader := RCLo_PrepareDropPart;
					sRunData.TDataLoader.eModule := LMP_TurnOverArm;
					eManagerStep := SP_RunStp15;
				END_IF
			SP_RunStp15:
				IF sRunData.sStatusLoader = RS_WaitRequest THEN
					IF sRunData.TDataLoader.eModule = LMP_TurnOverArm THEN
						sRunData.eCmdTurnOver := RCTO_TakePart;
					END_IF
					sRunData.eCmdLoader := RCLo_GivePart;
					eManagerStep := SP_RunStp16;
				END_IF
			SP_RunStp16:
				IF sRunData.sStatusLoader = RS_WaitRequest AND sRunData.sStatusTurnOver = RS_WaitRequest THEN
					eManagerStep := SP_RunStp20;
				END_IF
			SP_RunStp20: (* Unloading finish, proceed cleaning and turn over*)
				eRestartStep := SP_RunStp20;
				eRestartLoaderStep := SP_RunStp20;
				IF iPartOnProcess = 0 AND NOT bNeedNewPart THEN
					eManagerStep := SP_RunStp100;
				ELSE
					sRunData.eCmdLoader := RCLo_MoveToSafe;
					eManagerStep := SP_RunStp21;
				END_IF
			SP_RunStp21:
				IF sRunData.sStatusLoader = RS_WaitRequest THEN
					IF sRunData.TDataTurnOver.aTPartData[TO_Arm].bPartPresent THEN
						sRunData.eCmdTurnOver := RCTO_Turn;
					END_IF
					IF NOT bTableIsClean THEN
						sRunData.eCmdTable := RCT_Clean;
					END_IF
					eManagerStep := SP_RunStp22;
				END_IF
			SP_RunStp22: (*Cleaning Table and proceed turn over*)
				IF sRunData.sStatusTable = RS_WaitRequest  AND sRunData.sStatusTurnOver = RS_WaitRequest THEN
					bTableIsClean := TRUE;
					eManagerStep := SP_RunStp23;
				END_IF
			SP_RunStp23:
				eRestartStep := SP_RunStp23;
				eRestartLoaderStep := SP_RunStp26;
				IF sRunData.TDataTurnOver.aTPartData[TO_Fix].bPartPresent THEN
					bTableIsClean := FALSE;
					eManagerStep := SP_RunStp24;
				ELSE
					eManagerStep := SP_RunStp40; (* Skip *)
				END_IF
			SP_RunStp24: (* Move part from turn over *)
				sRunData.TDataLoader.eModule := LMP_TurnOverFix;
				sRunData.TDataLoader.eTaker := LH_Head2;
				sRunData.eCmdLoader := RCLo_PrepareTakePart;
				eManagerStep := SP_RunStp25;
			SP_RunStp25:
				IF sRunData.sStatusLoader = RS_WaitRequest THEN
					sRunData.eCmdLoader := RCLo_TakePart;
					sRunData.eCmdTurnOver := RCTO_GivePart;
					eManagerStep := SP_RunStp26;
				END_IF
			SP_RunStp26:
				IF sRunData.sStatusLoader = RS_WaitRequest AND sRunData.sStatusTurnOver = RS_WaitRequest THEN
					sRunData.eCmdLoader := RCLo_Cleaning;
					eManagerStep := SP_RunStp27;
				END_IF
			SP_RunStp27:
				IF sRunData.sStatusLoader = RS_WaitRequest THEN
					sRunData.TDataLoader.eModule := LMP_Table;
					sRunData.TDataLoader.iLayringPos := 1;
					sRunData.TDataLoader.iLayringOffsetPos := 0;
					sRunData.eCmdLoader := RCLo_PrepareDropPart;
					eManagerStep := SP_RunStp28;
				END_IF
			SP_RunStp28:
				IF sRunData.sStatusLoader = RS_WaitRequest THEN
					sRunData.eCmdLoader := RCLo_GivePart;
					sRunData.TDataTable.iGiveTakeLayeringPosition := sRunData.TDataLoader.iLayringPos;
					sRunData.TDataTable.iGiveTakeLayeringOffsetPosition := sRunData.TDataLoader.iLayringOffsetPos;
					sRunData.eCmdTable := RCT_TakePart;
					eManagerStep := SP_RunStp29;
				END_IF
			SP_RunStp29:
				IF sRunData.sStatusLoader = RS_WaitRequest AND sRunData.sStatusTable = RS_WaitRequest THEN
					(* Reject part if not correctly dropped *)
					IF sRunData.TDataLoader.aTPartData[LH_Head2].bPartPresent THEN
						eManagerStep := SP_RunStp30;
					ELSE
						eManagerStep := SP_RunStp40;
					END_IF
				END_IF
			SP_RunStp30:
				sRunData.TDataLoader.eModule := LMP_Reject;
				sRunData.eCmdLoader := RCLo_PrepareDropPart;
				eManagerStep := SP_RunStp15;
			SP_RunStp40: (* Load layering 1 *)
				eRestartStep := SP_RunStp40;
				eRestartLoaderStep := SP_RunStp42;
				IF bNeedNewPart AND NOT sRunData.TDataTable.aTPartData[0,0,sRunData.TDataTable.eTableSide].bPartPresent THEN
					bTableIsClean := FALSE;
					sRunData.TDataLoader.eModule := LMP_Lift1;
					sRunData.TDataLoader.eTaker := LH_Head1;
					sRunData.eCmdLoader := RCLo_PrepareTakePart;
					eManagerStep := SP_RunStp41;
				ELSE
					eManagerStep := SP_RunStp50; (* Skip *)
				END_IF
			SP_RunStp41:
				IF sRunData.sStatusLoader = RS_WaitRequest THEN
					sRunData.eCmdLoader := RCLo_TakePart;
					eManagerStep := SP_RunStp42;
				END_IF
			SP_RunStp42:
				IF sRunData.sStatusLoader = RS_WaitRequest THEN
					(* Check if a part was taken or not *)
					IF sRunData.TDataLoader.aTPartData[LH_Head1].bPartPresent THEN
						sRunData.TDataLoader.eModule := LMP_Table;
						sRunData.TDataLoader.iLayringPos := 0;
						sRunData.TDataLoader.iLayringOffsetPos := 0;
						sRunData.eCmdLoader := RCLo_PrepareDropPart;
						eManagerStep := SP_RunStp43;
					ELSE
						eManagerStep := SP_RunStp40;
					END_IF
				END_IF
			SP_RunStp43:
				IF sRunData.sStatusLoader = RS_WaitRequest THEN
					sRunData.eCmdLoader := RCLo_GivePart;
					sRunData.TDataTable.iGiveTakeLayeringPosition := sRunData.TDataLoader.iLayringPos;
					sRunData.TDataTable.iGiveTakeLayeringOffsetPosition := sRunData.TDataLoader.iLayringOffsetPos;
					sRunData.eCmdTable := RCT_TakePart;
					eManagerStep := SP_RunStp44;
				END_IF
			SP_RunStp44:
				IF sRunData.sStatusLoader = RS_WaitRequest AND  sRunData.sStatusTable = RS_WaitRequest  THEN
					(* Reject part if not correctly dropped *)
					IF sRunData.TDataLoader.aTPartData[LH_Head2].bPartPresent THEN
						eManagerStep := SP_RunStp30;
					ELSE
						eManagerStep := SP_RunStp50;
					END_IF
				END_IF
			SP_RunStp50: (* Launch loader to safe *)
				eRestartStep := SP_RunStp50;
				eRestartLoaderStep := SP_RunStp50;
				sRunData.eCmdLoader := RCLo_MoveToSafe;
				eManagerStep := SP_RunStp51;
			SP_RunStp51:
				IF sRunData.sStatusLoader = RS_WaitRequest AND bPearlingFinishOnTableSide THEN
					(* Pearling finish *)
					bReadyForPearling := FALSE;
					eManagerStep := SP_RunStp52;
				END_IF
			SP_RunStp52:
				eRestartStep := SP_RunStp53;
				eRestartLoaderStep := SP_RunStp53;
				sRunData.eCmdTable := RCT_TurnAndClean;
				eWorkingTableSide := ePearlingTableSide;
				eManagerStep := SP_RunStp53;
			SP_RunStp53: (*Turning Table *)
				IF sRunData.sStatusTable = RS_ProcessRequest2 THEN
					bReadyForPearling := TRUE;
					eManagerStep := SP_RunStp54;
				END_IF
			SP_RunStp54: (*Cleaning Table *)
				IF sRunData.sStatusTable = RS_WaitRequest AND sRunData.sStatusLoader = RS_WaitRequest  THEN
					bTableIsClean := TRUE;
					eManagerStep := SP_RunStp1;
				END_IF
			SP_RunStp100: (*End of recipe *)
				bReadyForPearling := FALSE;
				sRunData.eCmdLoader := RCLo_EndOfRecipe;
				eManagerStep := SP_RunStp101;
			SP_RunStp101: (*Loader in safe and lift in unload position *)
				IF sRunData.sStatusLoader = RS_WaitRequest  AND sRunData.sStatusPearling = RS_WaitRequest THEN
					eManagerStep := SP_RunStp0;
				END_IF
		END_CASE
	ELSE
		CASE eManagerStep OF
(* Running Step, Parts is TurnOver at begining *)
			SP_RunStp1:
				eRestartStep := SP_RunStp1;
				eRestartLoaderStep := SP_RunStp4;
				IF sRunData.TDataTable.aTPartData[1,0,sRunData.TDataTable.eTableSide].bPartPresent THEN
					bTableIsClean := FALSE;
					eManagerStep := SP_RunStp2;
				ELSE
					eManagerStep := SP_RunStp10; (* Skip *)
				END_IF
			SP_RunStp2: (* Unloading part on layering 1 *)
				sRunData.TDataLoader.eModule := LMP_Table;
				sRunData.TDataLoader.eTaker := LH_Head2;
				sRunData.TDataLoader.iLayringPos := 1;
				sRunData.TDataLoader.iLayringOffsetPos := 0;
				sRunData.eCmdLoader := RCLo_PrepareTakePart;
				eManagerStep := SP_RunStp3;
			SP_RunStp3:
				IF sRunData.sStatusLoader = RS_WaitRequest THEN
					sRunData.eCmdLoader := RCLo_TakePart;
					sRunData.TDataTable.iGiveTakeLayeringPosition := sRunData.TDataLoader.iLayringPos;
					sRunData.TDataTable.iGiveTakeLayeringOffsetPosition := sRunData.TDataLoader.iLayringOffsetPos;
					sRunData.eCmdTable := RCT_GivePart;
					eManagerStep := SP_RunStp4;
				END_IF
			SP_RunStp4:
				IF sRunData.sStatusLoader = RS_WaitRequest AND  sRunData.sStatusTable = RS_WaitRequest  THEN
					sRunData.eCmdLoader := RCLo_Cleaning;
					eManagerStep := SP_RunStp5;
				END_IF
			SP_RunStp5:
				IF sRunData.sStatusLoader = RS_WaitRequest  THEN
					IF sRunData.TDataLoader.aTPartData[LH_Head2].bToReject THEN
						sRunData.TDataLoader.eModule := LMP_Reject;
					ELSIF sProductionCmd.TRequestSample.Activate THEN
						sRunData.TDataLoader.eModule := LMP_Sample;
						sProductionCmd.TRequestSample.Activate := FALSE;
					ELSE
						sProductionCmd.TAutoSampling.iPeriodCnt := sProductionCmd.TAutoSampling.iPeriodCnt + 1;
						IF sProductionCmd.TAutoSampling.bEnable AND (sProductionCmd.TAutoSampling.iPeriodCnt >= (sProductionCmd.TAutoSampling.iPeriod - sProductionCmd.TAutoSampling.iBatchSize)) THEN
							sRunData.TDataLoader.eModule := LMP_Sample;
							sProductionCmd.TAutoSampling.iBatchCnt := sProductionCmd.TAutoSampling.iBatchCnt + 1;
							IF sProductionCmd.TAutoSampling.iBatchCnt >= sProductionCmd.TAutoSampling.iBatchSize THEN
								sProductionCmd.TAutoSampling.iBatchCnt := 0;
								sProductionCmd.TAutoSampling.iPeriodCnt := 0;
							END_IF
						ELSE
							sRunData.TDataLoader.eModule := LMP_Lift2;
						END_IF
					END_IF
					sRunData.eCmdLoader := RCLo_PrepareDropPart;
					eManagerStep := SP_RunStp6;
				END_IF
			SP_RunStp6:
				IF sRunData.sStatusLoader = RS_WaitRequest THEN
					sRunData.eCmdLoader := RCLo_GivePart;
					eManagerStep := SP_RunStp7;
				END_IF
			SP_RunStp7:
				IF sRunData.sStatusLoader = RS_WaitRequest THEN
					eManagerStep := SP_RunStp10;
				END_IF
			SP_RunStp10: (* Load Part on TurnOver *)
				eRestartStep := SP_RunStp10;
				eRestartLoaderStep := SP_RunStp12;
				IF bNeedNewPart AND NOT sRunData.TDataTurnOver.aTPartData[TO_Arm].bPartPresent AND NOT sRunData.TDataTurnOver.aTPartData[TO_Fix].bPartPresent THEN
					sRunData.TDataLoader.eModule := LMP_Lift1;
					sRunData.TDataLoader.eTaker := LH_Head1;
					sRunData.eCmdLoader := RCLo_PrepareTakePart;
					eManagerStep := SP_RunStp11;
				ELSE
					eManagerStep := SP_RunStp20; (* Skip *)
				END_IF
			SP_RunStp11:
				IF sRunData.sStatusLoader = RS_WaitRequest THEN
					sRunData.eCmdLoader := RCLo_TakePart;
					eManagerStep := SP_RunStp12;
				END_IF
			SP_RunStp12:
				IF sRunData.sStatusLoader = RS_WaitRequest THEN
					(* Check if a part was taken or not *)
					IF sRunData.TDataLoader.aTPartData[LH_Head1].bPartPresent THEN
						sRunData.eCmdLoader := RCLo_PrepareDropPart;
						sRunData.TDataLoader.eModule := LMP_TurnOverArm;
						eManagerStep := SP_RunStp13;
					ELSE
						eManagerStep := SP_RunStp10;
					END_IF
				END_IF
			SP_RunStp13:
				IF sRunData.sStatusLoader = RS_WaitRequest THEN
					IF sRunData.TDataLoader.eModule = LMP_TurnOverArm THEN
						sRunData.eCmdTurnOver := RCTO_TakePart;
					END_IF
					sRunData.eCmdLoader := RCLo_GivePart;
					eManagerStep := SP_RunStp14;
				END_IF
			SP_RunStp14:
				IF sRunData.sStatusLoader = RS_WaitRequest AND sRunData.sStatusTurnOver = RS_WaitRequest THEN
					eManagerStep := SP_RunStp20;
				END_IF
			SP_RunStp20: (* Unloading finish, proceed cleaning and turn over*)
				eRestartStep := SP_RunStp20;
				eRestartLoaderStep := SP_RunStp20;
				IF iPartOnProcess = 0 AND NOT bNeedNewPart THEN
					eManagerStep := SP_RunStp100;
				ELSE
					sRunData.eCmdLoader := RCLo_MoveToSafe;
					eManagerStep := SP_RunStp21;
				END_IF
			SP_RunStp21:
				IF sRunData.sStatusLoader = RS_WaitRequest THEN
					IF sRunData.TDataTurnOver.aTPartData[TO_Arm].bPartPresent THEN
						sRunData.eCmdTurnOver := RCTO_Turn;
					END_IF
					IF NOT bTableIsClean THEN
						sRunData.eCmdTable := RCT_Clean;
					END_IF
					eManagerStep := SP_RunStp22;
				END_IF
			SP_RunStp22: (*Cleaning Table and proceed turn over*)
				IF sRunData.sStatusTable = RS_WaitRequest  AND sRunData.sStatusTurnOver = RS_WaitRequest THEN
					bTableIsClean := TRUE;
					eManagerStep := SP_RunStp23;
				END_IF
			SP_RunStp23:
				eRestartStep := SP_RunStp23;
				eRestartLoaderStep := SP_RunStp26;
				IF sRunData.TDataTurnOver.aTPartData[TO_Fix].bPartPresent THEN
					bTableIsClean := FALSE;
					eManagerStep := SP_RunStp24;
				ELSE
					eManagerStep := SP_RunStp50; (* Skip *)
				END_IF
			SP_RunStp24: (* Move part from turn over *)
				sRunData.TDataLoader.eModule := LMP_TurnOverFix;
				sRunData.TDataLoader.eTaker := LH_Head2;
				sRunData.eCmdLoader := RCLo_PrepareTakePart;
				eManagerStep := SP_RunStp25;
			SP_RunStp25:
				IF sRunData.sStatusLoader = RS_WaitRequest THEN
					sRunData.eCmdLoader := RCLo_TakePart;
					sRunData.eCmdTurnOver := RCTO_GivePart;
					eManagerStep := SP_RunStp26;
				END_IF
			SP_RunStp26:
				IF sRunData.sStatusLoader = RS_WaitRequest AND sRunData.sStatusTurnOver = RS_WaitRequest THEN
					sRunData.TDataLoader.eModule := LMP_Table;
					sRunData.TDataLoader.iLayringPos := 1;
					sRunData.TDataLoader.iLayringOffsetPos := 0;
					sRunData.eCmdLoader := RCLo_PrepareDropPart;
					eManagerStep := SP_RunStp28;
				END_IF
			SP_RunStp28:
				IF sRunData.sStatusLoader = RS_WaitRequest THEN
					sRunData.eCmdLoader := RCLo_GivePart;
					sRunData.TDataTable.iGiveTakeLayeringPosition := sRunData.TDataLoader.iLayringPos;
					sRunData.TDataTable.iGiveTakeLayeringOffsetPosition := sRunData.TDataLoader.iLayringOffsetPos;
					sRunData.eCmdTable := RCT_TakePart;
					eManagerStep := SP_RunStp29;
				END_IF
			SP_RunStp29:
				IF sRunData.sStatusLoader = RS_WaitRequest AND sRunData.sStatusTable = RS_WaitRequest THEN
					(* Reject part if not correctly dropped *)
					IF sRunData.TDataLoader.aTPartData[LH_Head2].bPartPresent THEN
						eManagerStep := SP_RunStp30;
					ELSE
						eManagerStep := SP_RunStp50;
					END_IF
				END_IF
			SP_RunStp30:
				sRunData.TDataLoader.eModule := LMP_Reject;
				sRunData.eCmdLoader := RCLo_PrepareDropPart;
				eManagerStep := SP_RunStp13;
			SP_RunStp50: (* Launch loader to safe *)
				eRestartStep := SP_RunStp50;
				eRestartLoaderStep := SP_RunStp50;
				sRunData.eCmdLoader := RCLo_MoveToSafe;
				eManagerStep := SP_RunStp51;
			SP_RunStp51:
				IF sRunData.sStatusLoader = RS_WaitRequest AND bPearlingFinishOnTableSide THEN
					(* Pearling finish *)
					bReadyForPearling := FALSE;
					eManagerStep := SP_RunStp52;
				END_IF
			SP_RunStp52:
				eRestartStep := SP_RunStp53;
				eRestartLoaderStep := SP_RunStp53;
				sRunData.eCmdTable := RCT_TurnAndClean;
				eWorkingTableSide := ePearlingTableSide;
				eManagerStep := SP_RunStp53;
			SP_RunStp53: (*Turning Table *)
				IF sRunData.sStatusTable = RS_ProcessRequest2  THEN
					bReadyForPearling := TRUE;
					eManagerStep := SP_RunStp54;
				END_IF
			SP_RunStp54: (*Cleaning Table *)
				IF sRunData.sStatusTable = RS_WaitRequest AND  sRunData.sStatusLoader = RS_WaitRequest  THEN
					bTableIsClean := TRUE;
					eManagerStep := SP_RunStp1;
				END_IF
			SP_RunStp100: (*End of recipe *)
				bReadyForPearling := FALSE;
				sRunData.eCmdLoader := RCLo_EndOfRecipe;
				eManagerStep := SP_RunStp101;
			SP_RunStp101: (*Loader in safe and lift in unload position *)
				IF sRunData.sStatusLoader = RS_WaitRequest  AND sRunData.sStatusPearling = RS_WaitRequest THEN
					eManagerStep := SP_RunStp0;
				END_IF
		END_CASE
	END_IF
	IF bSimPearling AND  bReadyForPearling THEN
		IF sRunData.TDataTable.aTPartData[0,0,ePearlingTableSide].bPartPresent AND  sConfigFileData.asPearlingData[PS_SUS].THead[PH_Left].nNbOfPearls > 0 THEN
			sRunData.TDataTable.aTPartData[0,0,ePearlingTableSide].abPearlingDone[PH_Left,PS_SUS] := TRUE;
		END_IF
		IF sRunData.TDataTable.aTPartData[0,0,ePearlingTableSide].bPartPresent AND  sConfigFileData.asPearlingData[PS_SUS].THead[PH_Right].nNbOfPearls > 0 THEN
			sRunData.TDataTable.aTPartData[0,0,ePearlingTableSide].abPearlingDone[PH_Right,PS_SUS] := TRUE;
		END_IF
		IF sRunData.TDataTable.aTPartData[1,0,ePearlingTableSide].bPartPresent AND  sConfigFileData.asPearlingData[PS_SOUS].THead[PH_Left].nNbOfPearls > 0 THEN
			sRunData.TDataTable.aTPartData[1,0,ePearlingTableSide].abPearlingDone[PH_Left,PS_SOUS] := TRUE;
		END_IF
		IF sRunData.TDataTable.aTPartData[1,0,ePearlingTableSide].bPartPresent AND  sConfigFileData.asPearlingData[PS_SOUS].THead[PH_Right].nNbOfPearls > 0 THEN
			sRunData.TDataTable.aTPartData[1,0,ePearlingTableSide].abPearlingDone[PH_Right,PS_SOUS] := TRUE;
		END_IF
	ELSIF  NOT bSimPearling AND sRunData.sStatusPearling = RS_WaitRequest  AND  bReadyForPearling THEN
		(* Pearling does nothing, launch pearling if there is part to pearl *)
		sRunData.TDataPearling.abUseSpindle[PH_Left] := FALSE;
		sRunData.TDataPearling.abUseSpindle[PH_Right] := FALSE;
		IF 	sRunData.TDataTable.aTPartData[0,0,ePearlingTableSide].bPartPresent AND
			NOT sRunData.TDataTable.aTPartData[0,0,ePearlingTableSide].abPearlingDone[PH_Left,PS_SUS] AND
			sConfigFileData.asPearlingData[PS_SUS].THead[PH_Left].nNbOfPearls > 0 THEN
			(* Launch pearling on this part *)
			sRunData.TDataPearling.sPearlingData := sConfigFileData.asPearlingData[PS_SUS].THead[PH_Left];
			sRunData.TDataPearling.abUseSpindle[PH_Left] := TRUE;
			sRunData.TDataPearling.iLayringPos := 0;
			sRunData.TDataPearling.iLayringOffsetPos := 0;
			sRunData.TDataPearling.apsPartData[PH_Left] := ADR(sRunData.TDataTable.aTPartData[0,0,ePearlingTableSide]);
			sRunData.TDataPearling.bForceSharpenAfterPearling := sConfigFileData.asPearlingData[PS_SUS].THead[PH_Right].nNbOfPearls = 0;
			sRunData.eCmdPearling := RCP_Pearl;
		ELSIF sRunData.TDataTable.aTPartData[0,0,ePearlingTableSide].bPartPresent AND
			NOT sRunData.TDataTable.aTPartData[0,0,ePearlingTableSide].abPearlingDone[PH_Right,PS_SUS] AND
			sConfigFileData.asPearlingData[PS_SUS].THead[PH_Right].nNbOfPearls > 0 THEN
			(* Launch pearling on this part *)
			sRunData.TDataPearling.sPearlingData := sConfigFileData.asPearlingData[PS_SUS].THead[PH_Right];
			sRunData.TDataPearling.abUseSpindle[PH_Right] := TRUE;
			sRunData.TDataPearling.iLayringPos := 0;
			sRunData.TDataPearling.iLayringOffsetPos := 0;
			sRunData.TDataPearling.apsPartData[PH_Right] := ADR(sRunData.TDataTable.aTPartData[0,0,ePearlingTableSide]);
			sRunData.TDataPearling.bForceSharpenAfterPearling := TRUE;
			sRunData.eCmdPearling := RCP_Pearl;
		ELSIF 	sRunData.TDataTable.aTPartData[1,0,ePearlingTableSide].bPartPresent AND
			NOT sRunData.TDataTable.aTPartData[1,0,ePearlingTableSide].abPearlingDone[PH_Left,PS_SOUS] AND
			sConfigFileData.asPearlingData[PS_SOUS].THead[PH_Left].nNbOfPearls > 0 THEN
			(* Launch pearling on this part *)
			sRunData.TDataPearling.sPearlingData := sConfigFileData.asPearlingData[PS_SOUS].THead[PH_Left];
			sRunData.TDataPearling.abUseSpindle[PH_Left] := TRUE;
			sRunData.TDataPearling.iLayringPos := 1;
			sRunData.TDataPearling.iLayringOffsetPos := 0;
			sRunData.TDataPearling.apsPartData[PH_Left] := ADR(sRunData.TDataTable.aTPartData[1,0,ePearlingTableSide]);
			sRunData.TDataPearling.bForceSharpenAfterPearling := sConfigFileData.asPearlingData[PS_SOUS].THead[PH_Right].nNbOfPearls = 0;
			sRunData.eCmdPearling := RCP_Pearl;
		ELSIF sRunData.TDataTable.aTPartData[1,0,ePearlingTableSide].bPartPresent AND
			NOT sRunData.TDataTable.aTPartData[1,0,ePearlingTableSide].abPearlingDone[PH_Right,PS_SOUS] AND
			sConfigFileData.asPearlingData[PS_SOUS].THead[PH_Right].nNbOfPearls > 0 THEN
			(* Launch pearling on this part *)
			sRunData.TDataPearling.sPearlingData := sConfigFileData.asPearlingData[PS_SOUS].THead[PH_Right];
			sRunData.TDataPearling.abUseSpindle[PH_Right] := TRUE;
			sRunData.TDataPearling.iLayringPos := 1;
			sRunData.TDataPearling.iLayringOffsetPos := 0;
			sRunData.TDataPearling.apsPartData[PH_Right] := ADR(sRunData.TDataTable.aTPartData[1,0,ePearlingTableSide]);
			sRunData.TDataPearling.bForceSharpenAfterPearling := TRUE;
			sRunData.eCmdPearling := RCP_Pearl;
		END_IF
	END_IF

ELSIF sConfigFileData.bParallelProduction OR bLayeringWithTwoParts THEN

	IF sRunData.sStatusPearling <> RS_WaitRequest THEN
		bPearlingFinishOnTableSide := FALSE;
	ELSE
		bPearlingFinishOnTableSide := TRUE;
		IF bLayeringWithTwoParts THEN
			IF	   ( sRunData.TDataTable.aTPartData[0,0,ePearlingTableSide].bPartPresent AND NOT (sRunData.TDataTable.aTPartData[0,0,ePearlingTableSide].abPearlingDone[PH_Left,PS_SUS] OR sRunData.TDataTable.aTPartData[0,0,ePearlingTableSide].abPearlingDone[PH_Right,PS_SUS])) 
				OR ( sRunData.TDataTable.aTPartData[0,1,ePearlingTableSide].bPartPresent AND NOT (sRunData.TDataTable.aTPartData[0,1,ePearlingTableSide].abPearlingDone[PH_Left,PS_SUS] OR sRunData.TDataTable.aTPartData[0,1,ePearlingTableSide].abPearlingDone[PH_Right,PS_SUS])) 
				OR ( sRunData.TDataTable.aTPartData[1,0,ePearlingTableSide].bPartPresent AND NOT (sRunData.TDataTable.aTPartData[1,0,ePearlingTableSide].abPearlingDone[PH_Left,PS_SUS] OR sRunData.TDataTable.aTPartData[1,0,ePearlingTableSide].abPearlingDone[PH_Right,PS_SUS])) 
				OR ( sRunData.TDataTable.aTPartData[1,1,ePearlingTableSide].bPartPresent AND NOT (sRunData.TDataTable.aTPartData[1,1,ePearlingTableSide].abPearlingDone[PH_Left,PS_SUS] OR sRunData.TDataTable.aTPartData[1,1,ePearlingTableSide].abPearlingDone[PH_Right,PS_SUS])) 
				THEN
				bPearlingFinishOnTableSide := FALSE;
			END_IF
		ELSE
			IF	   ( sRunData.TDataTable.aTPartData[0,0,ePearlingTableSide].bPartPresent AND NOT (sRunData.TDataTable.aTPartData[0,0,ePearlingTableSide].abPearlingDone[PH_Left,PS_SUS] OR sRunData.TDataTable.aTPartData[0,0,ePearlingTableSide].abPearlingDone[PH_Right,PS_SUS])) 
				OR ( sRunData.TDataTable.aTPartData[1,0,ePearlingTableSide].bPartPresent AND NOT (sRunData.TDataTable.aTPartData[1,0,ePearlingTableSide].abPearlingDone[PH_Left,PS_SUS] OR sRunData.TDataTable.aTPartData[1,0,ePearlingTableSide].abPearlingDone[PH_Right,PS_SUS])) 
				THEN
				bPearlingFinishOnTableSide := FALSE;
			END_IF
		END_IF
	END_IF
	IF bUse103171OptimA1 THEN
		CASE eManagerStep OF
			SP_InitStp1:	(*Recovery, Drop plate if we have one*)
				sRunData.eCmdPearling := RCP_CheckSharpen;
				bReadyForPearling := FALSE;
				bTableIsClean := FALSE;
				IF sRunData.TDataLoader.bPlatePresent THEN
					sRunData.eCmdLoader := RCLo_SwitchPlate;
					eManagerStep := SP_InitStp2;
				ELSE
					eManagerStep := SP_InitStp3;
				END_IF
			SP_InitStp2: (* Switch plate done *)
				IF sRunData.sStatusLoader = RS_WaitRequest THEN
					eManagerStep := SP_InitStp3;
				END_IF
			SP_InitStp3: (* Do we need a table turn ? *)
				IF  sRunData.TDataTable.eTableSide <>  eWorkingTableSide THEN
					sRunData.eCmdTable := RCT_Turn;
					eManagerStep := SP_InitStp4;
				ELSE
					eManagerStep := SP_InitStp5;
				END_IF
			SP_InitStp4:
					IF sRunData.sStatusTable = RS_WaitRequest THEN
						eManagerStep := SP_InitStp5;
					END_IF
			SP_InitStp5:
				bReadyForPearling := TRUE;
				IF sRunData.TDataLoader.aTPartData[LH_Head1].bPartPresent THEN
					eManagerStep := eRestartLoaderStep;
				ELSE
					eManagerStep := eRestartStep;
				END_IF
	(* Running Step *)
			SP_RunStp1:
				sRunData.TDataLoader.iLayringOffsetPos := 0;
				sRunData.TDataTable.iGiveTakeLayeringOffsetPosition := sRunData.TDataLoader.iLayringOffsetPos;
				eRestartStep := SP_RunStp1;
				eRestartLoaderStep := SP_RunStp1;
				// Check if parts can be taken on table
				IF sRunData.TDataTable.aTPartData[0,0,sRunData.TDataTable.eTableSide].bPartPresent
						AND NOT sRunData.TDataLoader.aTPartData[0].bPartPresent THEN
					// Take the part on table with head1
					bTableIsClean := FALSE;
					sRunData.TDataLoader.eModule := LMP_Table;
					sRunData.TDataLoader.eTaker := LH_Head1;
					sRunData.TDataLoader.iLayringPos := 0;
					eManagerStep := SP_RunStp100;
				ELSIF sRunData.TDataTable.aTPartData[1,0,sRunData.TDataTable.eTableSide].bPartPresent
						AND NOT sRunData.TDataLoader.aTPartData[1].bPartPresent THEN
					// Take the part on table with head2
					bTableIsClean := FALSE;
					sRunData.TDataLoader.eModule := LMP_Table;
					sRunData.TDataLoader.eTaker := LH_Head2;
					sRunData.TDataLoader.iLayringPos := 1;
					eManagerStep := SP_RunStp100;
				ELSIF NOT sRunData.TDataLoader.aTPartData[0].bPartPresent 
						AND NOT sRunData.TDataLoader.aTPartData[1].bPartPresent THEN
					// Move loader to safe for cleaning and reload
					sRunData.eCmdLoader := RCLo_MoveToSafe;
					eManagerStep := SP_RunStp50;
				ELSE
					// Move loader to safe and drop part
					sRunData.eCmdLoader := RCLo_MoveToSafe;
					eManagerStep := SP_RunStp2;
				END_IF
			SP_RunStp2: // Drop parts and check table
				IF sRunData.sStatusLoader = RS_WaitRequest THEN
					// Check if table can be cleaned
					IF sRunData.sStatusTable = RS_WaitRequest
							AND NOT sRunData.TDataTable.aTPartData[0,0,sRunData.TDataTable.eTableSide].bPartPresent
							AND NOT sRunData.TDataTable.aTPartData[1,0,sRunData.TDataTable.eTableSide].bPartPresent 
							AND NOT bTableIsClean THEN
						// Clean the table
						sRunData.eCmdTable := RCT_Clean;
					END_IF
					// Check if part must be dropped
					IF sRunData.TDataLoader.aTPartData[0].bPartPresent THEN
						// Drop part on head 1
						sRunData.TDataLoader.eTaker := LH_Head1;
						eManagerStep := SP_RunStp200;
					ELSIF sRunData.TDataLoader.aTPartData[1].bPartPresent THEN
						// Drop part on head 2
						sRunData.TDataLoader.eTaker := LH_Head2;
						eManagerStep := SP_RunStp200;
					ELSIF sRunData.sStatusTable = RS_WaitRequest THEN
						// No more parts on head and table is clean
						bTableIsClean := TRUE;
						eManagerStep := SP_RunStp1;
					END_IF
				END_IF
	
